   1:  PR[91,2] = PR[90,2] + 11.921;
   1:L PR[91] R[100]mm/sec CNT100;
   1:  PR[91,1] = PR[90,1] + -55.817;
   1:  PR[91,2] = PR[90,2] + 11.419;
   1:L PR[91] R[100]mm/sec CNT100;
   1:  PR[91,1] = PR[90,1] + -55.517;
   1:  PR[91,2] = PR[90,2] + 10.784;
   1:L PR[91] R[100]mm/sec CNT100;
   1:  PR[91,1] = PR[90,1] + -55.501;
   1:  PR[91,2] = PR[90,2] + 10.726;
   1:L PR[91] R[100]mm/sec CNT100;
   1:  PR[91,1] = PR[90,1] + -54.925;
   1:  PR[91,2] = PR[90,2] + 10.182;
   1:L PR[91] R[100]mm/sec CNT100;
   1:  PR[91,1] = PR[90,1] + -54.832;
   1:  PR[91,2] = PR[90,2] + 9.653;
   1:L PR[91] R[100]mm/sec CNT100;
   1:  PR[91,1] = PR[90,1] + -54.444;
   1:  PR[91,2] = PR[90,2] + 8.648;
   1:L PR[91] R[100]mm/sec CNT100;
   1:  PR[91,1] = PR[90,1] + -54.411;
   1:  PR[91,2] = PR[90,2] + 8.471;
   1:L PR[91] R[100]mm/sec CNT100;
   1:  PR[91,1] = PR[90,1] + -53.977;
   1:  PR[91,2] = PR[90,2] + 7.812;
   1:L PR[91] R[100]mm/sec CNT100;
   1:  PR[91,1] = PR[90,1] + -53.950;
   1:  PR[91,2] = PR[90,2] + 7.562;
   1:L PR[91] R[100]mm/sec CNT100;
   1:  PR[91,1] = PR[90,1] + -53.710;
   1:  PR[91,2] = PR[90,2] + 6.887;
   1:L PR[91] R[100]mm/sec CNT100;
   1:  PR[91,1] = PR[90,1] + -53.581;
   1:  PR[91,2] = PR[90,2] + 5.901;
   1:L PR[91] R[100]mm/sec CNT100;
   1:  PR[91,1] = PR[90,1] + -53.473;
   1:  PR[91,2] = PR[90,2] + 5.417;
   1:L PR[91] R[100]mm/sec CNT100;
   1:  PR[91,1] = PR[90,1] + -53.442;
   1:  PR[91,2] = PR[90,2] + 4.966;
   1:L PR[91] R[100]mm/sec CNT100;
   1:  PR[91,1] = PR[90,1] + -53.316;
   1:  PR[91,2] = PR[90,2] + 4.379;
   1:L PR[91] R[100]mm/sec CNT100;
   1:  PR[91,1] = PR[90,1] + -53.302;
   1:  PR[91,2] = PR[90,2] + 4.009;
   1:L PR[91] R[100]mm/sec CNT100;
   1:  PR[91,1] = PR[90,1] + -53.207;
   1:  PR[91,2] = PR[90,2] + 3.307;
   1:L PR[91] R[100]mm/sec CNT100;
   1:  PR[91,1] = PR[90,1] + -53.165;
   1:  PR[91,2] = PR[90,2] + 2.173;
   1:L PR[91] R[100]mm/sec CNT100;
   1:  PR[91,1] = PR[90,1] + -53.173;
   1:  PR[91,2] = PR[90,2] + 1.917;
   1:L PR[91] R[100]mm/sec CNT100;
   1:  PR[91,1] = PR[90,1] + -53.240;
   1:  PR[91,2] = PR[90,2] + 0.760;
   1:L PR[91] R[100]mm/sec CNT100;
   1:  PR[91,1] = PR[90,1] + -53.353;
   1:  PR[91,2] = PR[90,2] + -0.035;
   1:L PR[91] R[100]mm/sec CNT100;
   1:  PR[91,1] = PR[90,1] + -53.396;
   1:  PR[91,2] = PR[90,2] + -0.473;
   1:L PR[91] R[100]mm/sec CNT100;
   1:  PR[91,1] = PR[90,1] + -53.528;
   1:  PR[91,2] = PR[90,2] + -1.127;
   1:L PR[91] R[100]mm/sec CNT100;
   1:  PR[91,1] = PR[90,1] + -53.622;
   1:  PR[91,2] = PR[90,2] + -1.751;
   1:L PR[91] R[100]mm/sec CNT100;
   1:  PR[91,1] = PR[90,1] + -53.730;
   1:  PR[91,2] = PR[90,2] + -2.252;
   1:L PR[91] R[100]mm/sec CNT100;
   1:  PR[91,1] = PR[90,1] + -54.082;
   1:  PR[91,2] = PR[90,2] + -3.438;
   1:L PR[91] R[100]mm/sec CNT100;
   1:  PR[91,1] = PR[90,1] + -54.607;
   1:  PR[91,2] = PR[90,2] + -4.510;
   1:L PR[91] R[100]mm/sec CNT100;
   1:  PR[91,1] = PR[90,1] + -55.042;
   1:  PR[91,2] = PR[90,2] + -5.607;
   1:L PR[91] R[100]mm/sec CNT100;
   1:  PR[92] = PR[91];
   1:  PR[92,3] = PR[92,3] + R[101];
   1:J PR[92] R[102]% CNT100;
   1:  PR[91,1] = PR[90,1] + -50.789;
   1:  PR[91,2] = PR[90,2] + -0.113;
   1:  PR[92] = PR[91];
   1:  PR[92,3] = PR[92,3] + R[101];
   1:J PR[92] R[102]% CNT100;
   1:L PR[91] 100mm/sec CNT100 RampTo R[100];
   1:  PR[91,1] = PR[90,1] + -43.436;
   1:  PR[91,2] = PR[90,2] + 7.239;
   1:L PR[91] R[100]mm/sec CNT100;
   1:  PR[91,1] = PR[90,1] + -43.681;
   1:  PR[91,2] = PR[90,2] + 7.608;
   1:L PR[91] R[100]mm/sec CNT100;
   1:  PR[91,1] = PR[90,1] + -44.697;
   1:  PR[91,2] = PR[90,2] + 8.101;
   1:L PR[91] R[100]mm/sec CNT100;
   1:  PR[91,1] = PR[90,1] + -45.153;
   1:  PR[91,2] = PR[90,2] + 9.127;
   1:L PR[91] R[100]mm/sec CNT100;
   1:  PR[91,1] = PR[90,1] + -45.528;
   1:  PR[91,2] = PR[90,2] + 9.390;
   1:L PR[91] R[100]mm/sec CNT100;
   1:  PR[91,1] = PR[90,1] + -50.750;
   1:  PR[91,2] = PR[90,2] + 4.168;
   1:L PR[91] R[100]mm/sec CNT100;
   1:  PR[91,1] = PR[90,1] + -50.758;
   1:  PR[91,2] = PR[90,2] + 4.229;
   1:L PR[91] R[100]mm/sec CNT100;
   1:  PR[91,1] = PR[90,1] + -50.777;
   1:  PR[91,2] = PR[90,2] + 4.699;
   1:L PR[91] R[100]mm/sec CNT100;
   1:  PR[91,1] = PR[90,1] + -50.910;
   1:  PR[91,2] = PR[90,2] + 5.321;
   1:L PR[91] R[100]mm/sec CNT100;
   1:  PR[91,1] = PR[90,1] + -50.942;
   1:  PR[91,2] = PR[90,2] + 5.783;
   1:L PR[91] R[100]mm/sec CNT100;
   1:  PR[91,1] = PR[90,1] + -51.067;
   1:  PR[91,2] = PR[90,2] + 6.345;
   1:L PR[91] R[100]mm/sec CNT100;
   1:  PR[91,1] = PR[90,1] + -51.216;
   1:  PR[91,2] = PR[90,2] + 7.487;
   1:L PR[91] R[100]mm/sec CNT100;
   1:  PR[91,1] = PR[90,1] + -51.337;
   1:  PR[91,2] = PR[90,2] + 7.824;
   1:L PR[91] R[100]mm/sec CNT100;
   1:  PR[91,1] = PR[90,1] + -47.237;
   1:  PR[91,2] = PR[90,2] + 11.924;
   1:L PR[91] R[100]mm/sec CNT100;
   1:  PR[91,1] = PR[90,1] + -47.264;
   1:  PR[91,2] = PR[90,2] + 11.958;
   1:L PR[91] R[100]mm/sec CNT100;
   1:  PR[91,1] = PR[90,1] + -47.506;
   1:  PR[91,2] = PR[90,2] + 12.558;
   1:L PR[91] R[100]mm/sec CNT100;
   1:  PR[91,1] = PR[90,1] + -47.796;
   1:  PR[91,2] = PR[90,2] + 12.828;
   1:L PR[91] R[100]mm/sec CNT100;
   1:  PR[91,1] = PR[90,1] + -48.396;
   1:  PR[91,2] = PR[90,2] + 14.064;
   1:L PR[91] R[100]mm/sec CNT100;
   1:  PR[91,1] = PR[90,1] + -48.437;
   1:  PR[91,2] = PR[90,2] + 14.137;
   1:L PR[91] R[100]mm/sec CNT100;
   1:  PR[91,1] = PR[90,1] + -48.855;
   1:  PR[91,2] = PR[90,2] + 14.549;
   1:L PR[91] R[100]mm/sec CNT100;
   1:  PR[91,1] = PR[90,1] + -52.468;
   1:  PR[91,2] = PR[90,2] + 10.936;
   1:L PR[91] R[100]mm/sec CNT100;
   1:  PR[91,1] = PR[90,1] + -52.558;
   1:  PR[91,2] = PR[90,2] + 11.455;
   1:L PR[91] R[100]mm/sec CNT100;
   1:  PR[91,1] = PR[90,1] + -53.380;
   1:  PR[91,2] = PR[90,2] + 12.230;
   1:L PR[91] R[100]mm/sec CNT100;
   1:  PR[91,1] = PR[90,1] + -53.611;
   1:  PR[91,2] = PR[90,2] + 12.720;
   1:L PR[91] R[100]mm/sec CNT100;
   1:  PR[91,1] = PR[90,1] + -53.815;
   1:  PR[91,2] = PR[90,2] + 13.003;
   1:L PR[91] R[100]mm/sec CNT100;
   1:  PR[91,1] = PR[90,1] + -53.874;
   1:  PR[91,2] = PR[90,2] + 13.251;
   1:L PR[91] R[100]mm/sec CNT100;
   1:  PR[91,1] = PR[90,1] + -54.126;
   1:  PR[91,2] = PR[90,2] + 13.521;
   1:L PR[91] R[100]mm/sec CNT100;
   1:  PR[91,1] = PR[90,1] + -50.744;
   1:  PR[91,2] = PR[90,2] + 16.902;
   1:L PR[91] R[100]mm/sec CNT100;
   1:  PR[91,1] = PR[90,1] + -50.969;
   1:  PR[91,2] = PR[90,2] + 17.094;
   1:L PR[91] R[100]mm/sec CNT100;
   1:  PR[91,1] = PR[90,1] + -51.043;
   1:  PR[91,2] = PR[90,2] + 17.364;
   1:L PR[91] R[100]mm/sec CNT100;
   1:  PR[91,1] = PR[90,1] + -51.287;
   1:  PR[91,2] = PR[90,2] + 17.641;
   1:L PR[91] R[100]mm/sec CNT100;
   1:  PR[91,1] = PR[90,1] + -51.665;
   1:  PR[91,2] = PR[90,2] + 17.995;
   1:L PR[91] R[100]mm/sec CNT100;
   1:  PR[91,1] = PR[90,1] + -51.670;
   1:  PR[91,2] = PR[90,2] + 17.996;
   1:L PR[91] R[100]mm/sec CNT100;
   1:  PR[91,1] = PR[90,1] + -51.696;
   1:  PR[91,2] = PR[90,2] + 18.024;
   1:L PR[91] R[100]mm/sec CNT100;
   1:  PR[91,1] = PR[90,1] + -51.866;
   1:  PR[91,2] = PR[90,2] + 18.183;
   1:L PR[91] R[100]mm/sec CNT100;
   1:  PR[91,1] = PR[90,1] + -51.876;
   1:  PR[91,2] = PR[90,2] + 18.217;
   1:L PR[91] R[100]mm/sec CNT100;
   1:  PR[91,1] = PR[90,1] + -52.216;
   1:  PR[91,2] = PR[90,2] + 18.582;
   1:L PR[91] R[100]mm/sec CNT100;
   1:  PR[91,1] = PR[90,1] + -52.518;
   1:  PR[91,2] = PR[90,2] + 18.855;
   1:L PR[91] R[100]mm/sec CNT100;
   1:  PR[91,1] = PR[90,1] + -52.726;
   1:  PR[91,2] = PR[90,2] + 18.913;
   1:L PR[91] R[100]mm/sec CNT100;
   1:  PR[91,1] = PR[90,1] + -52.842;
   1:  PR[91,2] = PR[90,2] + 19.047;
   1:L PR[91] R[100]mm/sec CNT100;
   1:  PR[91,1] = PR[90,1] + -55.983;
   1:  PR[91,2] = PR[90,2] + 15.906;
   1:L PR[91] R[100]mm/sec CNT100;
   1:  PR[91,1] = PR[90,1] + -56.289;
   1:  PR[91,2] = PR[90,2] + 16.681;
   1:L PR[91] R[100]mm/sec CNT100;
   1:  PR[91,1] = PR[90,1] + -57.214;
   1:  PR[91,2] = PR[90,2] + 16.993;
   1:L PR[91] R[100]mm/sec CNT100;
   1:  PR[91,1] = PR[90,1] + -57.569;
   1:  PR[91,2] = PR[90,2] + 17.819;
   1:L PR[91] R[100]mm/sec CNT100;
   1:  PR[91,1] = PR[90,1] + -58.171;
   1:  PR[91,2] = PR[90,2] + 17.960;
   1:L PR[91] R[100]mm/sec CNT100;
   1:  PR[91,1] = PR[90,1] + -55.218;
   1:  PR[91,2] = PR[90,2] + 20.914;
   1:L PR[91] R[100]mm/sec CNT100;
   1:  PR[91,1] = PR[90,1] + -55.714;
   1:  PR[91,2] = PR[90,2] + 21.543;
   1:L PR[91] R[100]mm/sec CNT100;
   1:  PR[91,1] = PR[90,1] + -56.038;
   1:  PR[91,2] = PR[90,2] + 21.710;
   1:L PR[91] R[100]mm/sec CNT100;
   1:  PR[91,1] = PR[90,1] + -56.949;
   1:  PR[91,2] = PR[90,2] + 22.456;
   1:L PR[91] R[100]mm/sec CNT100;
   1:  PR[91,1] = PR[90,1] + -57.691;
   1:  PR[91,2] = PR[90,2] + 22.684;
   1:L PR[91] R[100]mm/sec CNT100;
   1:  PR[91,1] = PR[90,1] + -60.944;
   1:  PR[91,2] = PR[90,2] + 19.430;
   1:L PR[91] R[100]mm/sec CNT100;
   1:  PR[91,1] = PR[90,1] + -61.398;
   1:  PR[91,2] = PR[90,2] + 19.542;
   1:L PR[91] R[100]mm/sec CNT100;
   1:  PR[91,1] = PR[90,1] + -62.090;
   1:  PR[91,2] = PR[90,2] + 19.949;
   1:L PR[91] R[100]mm/sec CNT100;
   1:  PR[91,1] = PR[90,1] + -62.103;
   1:  PR[91,2] = PR[90,2] + 19.952;
   1:L PR[91] R[100]mm/sec CNT100;
   1:  PR[91,1] = PR[90,1] + -62.896;
   1:  PR[91,2] = PR[90,2] + 20.448;
   1:L PR[91] R[100]mm/sec CNT100;
   1:  PR[91,1] = PR[90,1] + -63.760;
   1:  PR[91,2] = PR[90,2] + 20.570;
   1:L PR[91] R[100]mm/sec CNT100;
   1:  PR[91,1] = PR[90,1] + -63.989;
   1:  PR[91,2] = PR[90,2] + 20.627;
   1:L PR[91] R[100]mm/sec CNT100;
   1:  PR[91,1] = PR[90,1] + -60.295;
   1:  PR[91,2] = PR[90,2] + 24.322;
   1:L PR[91] R[100]mm/sec CNT100;
   1:  PR[91,1] = PR[90,1] + -60.361;
   1:  PR[91,2] = PR[90,2] + 24.345;
   1:L PR[91] R[100]mm/sec CNT100;
   1:  PR[91,1] = PR[90,1] + -60.751;
   1:  PR[91,2] = PR[90,2] + 24.518;
   1:L PR[91] R[100]mm/sec CNT100;
   1:  PR[91,1] = PR[90,1] + -61.339;
   1:  PR[91,2] = PR[90,2] + 24.637;
   1:L PR[91] R[100]mm/sec CNT100;
   1:  PR[91,1] = PR[90,1] + -61.953;
   1:  PR[91,2] = PR[90,2] + 25.130;
   1:L PR[91] R[100]mm/sec CNT100;
   1:  PR[91,1] = PR[90,1] + -62.138;
   1:  PR[91,2] = PR[90,2] + 25.198;
   1:L PR[91] R[100]mm/sec CNT100;
   1:  PR[91,1] = PR[90,1] + -62.374;
   1:  PR[91,2] = PR[90,2] + 25.259;
   1:L PR[91] R[100]mm/sec CNT100;
   1:  PR[91,1] = PR[90,1] + -62.977;
   1:  PR[91,2] = PR[90,2] + 25.363;
   1:L PR[91] R[100]mm/sec CNT100;
   1:  PR[91,1] = PR[90,1] + -63.330;
   1:  PR[91,2] = PR[90,2] + 25.530;
   1:L PR[91] R[100]mm/sec CNT100;
   1:  PR[91,1] = PR[90,1] + -67.437;
   1:  PR[91,2] = PR[90,2] + 21.422;
   1:L PR[91] R[100]mm/sec CNT100;
   1:  PR[91,1] = PR[90,1] + -68.015;
   1:  PR[91,2] = PR[90,2] + 21.510;
   1:L PR[91] R[100]mm/sec CNT100;
   1:  PR[91,1] = PR[90,1] + -69.314;
   1:  PR[91,2] = PR[90,2] + 21.578;
   1:L PR[91] R[100]mm/sec CNT100;
   1:  PR[91,1] = PR[90,1] + -70.819;
   1:  PR[91,2] = PR[90,2] + 21.550;
   1:L PR[91] R[100]mm/sec CNT100;
   1:  PR[91,1] = PR[90,1] + -71.638;
   1:  PR[91,2] = PR[90,2] + 21.464;
   1:L PR[91] R[100]mm/sec CNT100;
   1:  PR[91,1] = PR[90,1] + -66.662;
   1:  PR[91,2] = PR[90,2] + 26.440;
   1:L PR[91] R[100]mm/sec CNT100;
   1:  PR[91,1] = PR[90,1] + -67.388;
   1:  PR[91,2] = PR[90,2] + 26.622;
   1:L PR[91] R[100]mm/sec CNT100;
   1:  PR[91,1] = PR[90,1] + -67.504;
   1:  PR[91,2] = PR[90,2] + 26.666;
   1:L PR[91] R[100]mm/sec CNT100;
   1:  PR[91,1] = PR[90,1] + -67.813;
   1:  PR[91,2] = PR[90,2] + 26.733;
   1:L PR[91] R[100]mm/sec CNT100;
   1:  PR[91,1] = PR[90,1] + -67.891;
   1:  PR[91,2] = PR[90,2] + 26.736;
   1:L PR[91] R[100]mm/sec CNT100;
   1:  PR[91,1] = PR[90,1] + -68.520;
   1:  PR[91,2] = PR[90,2] + 26.812;
   1:L PR[91] R[100]mm/sec CNT100;
   1:  PR[91,1] = PR[90,1] + -69.240;
   1:  PR[91,2] = PR[90,2] + 26.839;
   1:L PR[91] R[100]mm/sec CNT100;
   1:  PR[91,1] = PR[90,1] + -70.426;
   1:  PR[91,2] = PR[90,2] + 26.834;
   1:L PR[91] R[100]mm/sec CNT100;
   1:  PR[91,1] = PR[90,1] + -70.517;
   1:  PR[91,2] = PR[90,2] + 26.828;
   1:L PR[91] R[100]mm/sec CNT100;
   1:  PR[91,1] = PR[90,1] + -77.438;
   1:  PR[91,2] = PR[90,2] + 19.907;
   1:L PR[91] R[100]mm/sec CNT100;
   1:  PR[92] = PR[91];
   1:  PR[92,3] = PR[92,3] + R[101];
   1:J PR[92] R[102]% CNT100;
   1:  PR[91,1] = PR[90,1] + -91.029;
   1:  PR[91,2] = PR[90,2] + 44.499;
   1:  PR[92] = PR[91];
   1:  PR[92,3] = PR[92,3] + R[101];
   1:J PR[92] R[102]% CNT100;
   1:L PR[91] 100mm/sec CNT100 RampTo R[100];
   1:  PR[91,1] = PR[90,1] + -94.000;
   1:  PR[91,2] = PR[90,2] + 41.528;
   1:L PR[91] R[100]mm/sec CNT100;
   1:  PR[91,1] = PR[90,1] + -94.012;
   1:  PR[91,2] = PR[90,2] + 41.407;
   1:L PR[91] R[100]mm/sec CNT100;
   1:  PR[91,1] = PR[90,1] + -94.020;
   1:  PR[91,2] = PR[90,2] + 40.590;
   1:L PR[91] R[100]mm/sec CNT100;
   1:  PR[91,2] = PR[90,2] + 37.266;
   1:L PR[91] R[100]mm/sec CNT100;
   1:  PR[91,1] = PR[90,1] + -88.734;
   1:  PR[91,2] = PR[90,2] + 42.552;
   1:L PR[91] R[100]mm/sec CNT100;
   1:  PR[91,1] = PR[90,1] + -88.492;
   1:  PR[91,2] = PR[90,2] + 41.711;
   1:L PR[91] R[100]mm/sec CNT100;
   1:  PR[91,1] = PR[90,1] + -88.476;
   1:  PR[91,2] = PR[90,2] + 41.569;
   1:L PR[91] R[100]mm/sec CNT100;
   1:  PR[91,1] = PR[90,1] + -88.460;
   1:  PR[91,2] = PR[90,2] + 40.579;
   1:L PR[91] R[100]mm/sec CNT100;
   1:  PR[91,2] = PR[90,2] + 38.583;
   1:L PR[91] R[100]mm/sec CNT100;
   1:  PR[91,1] = PR[90,1] + -94.020;
   1:  PR[91,2] = PR[90,2] + 33.023;
   1:L PR[91] R[100]mm/sec CNT100;
   1:  PR[91,2] = PR[90,2] + 28.780;
   1:L PR[91] R[100]mm/sec CNT100;
   1:  PR[91,1] = PR[90,1] + -88.459;
   1:  PR[91,2] = PR[90,2] + 34.341;
   1:L PR[91] R[100]mm/sec CNT100;
   1:  PR[91,2] = PR[90,2] + 30.473;
   1:L PR[91] R[100]mm/sec CNT100;
   1:  PR[91,1] = PR[90,1] + -88.455;
   1:  PR[91,2] = PR[90,2] + 30.103;
   1:L PR[91] R[100]mm/sec CNT100;
   1:  PR[91,1] = PR[90,1] + -94.020;
   1:  PR[91,2] = PR[90,2] + 24.538;
   1:L PR[91] R[100]mm/sec CNT100;
   1:  PR[91,2] = PR[90,2] + 20.295;
   1:L PR[91] R[100]mm/sec CNT100;
   1:  PR[91,1] = PR[90,1] + -88.039;
   1:  PR[91,2] = PR[90,2] + 26.276;
   1:L PR[91] R[100]mm/sec CNT100;
   1:  PR[91,1] = PR[90,1] + -87.860;
   1:  PR[91,2] = PR[90,2] + 25.830;
   1:L PR[91] R[100]mm/sec CNT100;
   1:  PR[91,1] = PR[90,1] + -86.695;
   1:  PR[91,2] = PR[90,2] + 23.389;
   1:L PR[91] R[100]mm/sec CNT100;
   1:  PR[91,1] = PR[90,1] + -86.685;
   1:  PR[91,2] = PR[90,2] + 23.387;
   1:L PR[91] R[100]mm/sec CNT100;
   1:  PR[91,1] = PR[90,1] + -94.020;
   1:  PR[91,2] = PR[90,2] + 16.053;
   1:L PR[91] R[100]mm/sec CNT100;
   1:  PR[91,2] = PR[90,2] + 11.810;
   1:L PR[91] R[100]mm/sec CNT100;
   1:  PR[91,1] = PR[90,1] + -82.746;
   1:  PR[91,2] = PR[90,2] + 23.084;
   1:L PR[91] R[100]mm/sec CNT100;
   1:  PR[91,1] = PR[90,1] + -81.038;
   1:  PR[91,2] = PR[90,2] + 23.676;
   1:L PR[91] R[100]mm/sec CNT100;
   1:  PR[91,1] = PR[90,1] + -79.810;
   1:  PR[91,2] = PR[90,2] + 24.363;
   1:L PR[91] R[100]mm/sec CNT100;
   1:  PR[91,1] = PR[90,1] + -78.890;
   1:  PR[91,2] = PR[90,2] + 24.772;
   1:L PR[91] R[100]mm/sec CNT100;
   1:  PR[91,1] = PR[90,1] + -78.115;
   1:  PR[91,2] = PR[90,2] + 25.160;
   1:L PR[91] R[100]mm/sec CNT100;
   1:  PR[91,1] = PR[90,1] + -77.291;
   1:  PR[91,2] = PR[90,2] + 25.407;
   1:L PR[91] R[100]mm/sec CNT100;
   1:  PR[91,1] = PR[90,1] + -76.346;
   1:  PR[91,2] = PR[90,2] + 25.776;
   1:L PR[91] R[100]mm/sec CNT100;
   1:  PR[91,1] = PR[90,1] + -76.324;
   1:  PR[91,2] = PR[90,2] + 25.787;
   1:L PR[91] R[100]mm/sec CNT100;
   1:  PR[91,1] = PR[90,1] + -75.661;
   1:  PR[91,2] = PR[90,2] + 26.005;
   1:L PR[91] R[100]mm/sec CNT100;
   1:  PR[91,1] = PR[90,1] + -75.568;
   1:  PR[91,2] = PR[90,2] + 26.019;
   1:L PR[91] R[100]mm/sec CNT100;
   1:  PR[91,1] = PR[90,1] + -94.020;
   1:  PR[91,2] = PR[90,2] + 7.568;
   1:L PR[91] R[100]mm/sec CNT100;
   1:  PR[91,1] = PR[90,1] + -94.019;
   1:  PR[91,2] = PR[90,2] + 3.325;
   1:L PR[91] R[100]mm/sec CNT100;
   1:  PR[91,1] = PR[90,1] + -87.134;
   1:  PR[91,2] = PR[90,2] + 10.211;
   1:L PR[91] R[100]mm/sec CNT100;
   1:  PR[91,1] = PR[90,1] + -87.246;
   1:  PR[91,2] = PR[90,2] + 9.982;
   1:L PR[91] R[100]mm/sec CNT100;
   1:  PR[91,1] = PR[90,1] + -87.849;
   1:  PR[91,2] = PR[90,2] + 8.500;
   1:L PR[91] R[100]mm/sec CNT100;
   1:  PR[91,1] = PR[90,1] + -88.076;
   1:  PR[91,2] = PR[90,2] + 7.623;
   1:L PR[91] R[100]mm/sec CNT100;
   1:  PR[91,1] = PR[90,1] + -88.169;
   1:  PR[91,2] = PR[90,2] + 7.136;
   1:L PR[91] R[100]mm/sec CNT100;
   1:  PR[91,1] = PR[90,1] + -88.449;
   1:  PR[91,2] = PR[90,2] + 6.125;
   1:L PR[91] R[100]mm/sec CNT100;
   1:  PR[91,1] = PR[90,1] + -88.473;
   1:  PR[91,2] = PR[90,2] + 5.861;
   1:L PR[91] R[100]mm/sec CNT100;
   1:  PR[91,1] = PR[90,1] + -88.707;
   1:  PR[91,2] = PR[90,2] + 4.884;
   1:L PR[91] R[100]mm/sec CNT100;
   1:  PR[91,1] = PR[90,1] + -88.766;
   1:  PR[91,2] = PR[90,2] + 4.336;
   1:L PR[91] R[100]mm/sec CNT100;
   1:  PR[91,1] = PR[90,1] + -93.775;
   1:  PR[91,2] = PR[90,2] + -0.673;
   1:L PR[91] R[100]mm/sec CNT100;
   1:  PR[91,1] = PR[90,1] + -93.743;
   1:  PR[91,2] = PR[90,2] + -0.817;
   1:L PR[91] R[100]mm/sec CNT100;
   1:  PR[91,1] = PR[90,1] + -93.466;
   1:  PR[91,2] = PR[90,2] + -2.169;
   1:L PR[91] R[100]mm/sec CNT100;
   1:  PR[91,1] = PR[90,1] + -93.454;
   1:  PR[91,2] = PR[90,2] + -2.408;
   1:L PR[91] R[100]mm/sec CNT100;
   1:  PR[91,1] = PR[90,1] + -93.353;
   1:  PR[91,2] = PR[90,2] + -2.936;
   1:L PR[91] R[100]mm/sec CNT100;
   1:  PR[91,1] = PR[90,1] + -93.260;
   1:  PR[91,2] = PR[90,2] + -3.724;
   1:L PR[91] R[100]mm/sec CNT100;
   1:  PR[91,1] = PR[90,1] + -93.149;
   1:  PR[91,2] = PR[90,2] + -4.167;
   1:L PR[91] R[100]mm/sec CNT100;
   1:  PR[91,1] = PR[90,1] + -93.138;
   1:  PR[91,2] = PR[90,2] + -4.257;
   1:L PR[91] R[100]mm/sec CNT100;
   1:  PR[91,1] = PR[90,1] + -93.131;
   1:  PR[91,2] = PR[90,2] + -4.272;
   1:L PR[91] R[100]mm/sec CNT100;
   1:  PR[91,1] = PR[90,1] + -88.764;
   1:  PR[91,2] = PR[90,2] + 0.096;
   1:L PR[91] R[100]mm/sec CNT100;
   1:  PR[91,1] = PR[90,1] + -88.650;
   1:  PR[91,2] = PR[90,2] + -0.773;
   1:L PR[91] R[100]mm/sec CNT100;
   1:  PR[91,1] = PR[90,1] + -88.448;
   1:  PR[91,2] = PR[90,2] + -1.417;
   1:L PR[91] R[100]mm/sec CNT100;
   1:  PR[91,1] = PR[90,1] + -88.428;
   1:  PR[91,2] = PR[90,2] + -1.723;
   1:L PR[91] R[100]mm/sec CNT100;
   1:  PR[91,1] = PR[90,1] + -88.200;
   1:  PR[91,2] = PR[90,2] + -2.336;
   1:L PR[91] R[100]mm/sec CNT100;
   1:  PR[91,1] = PR[90,1] + -88.175;
   1:  PR[91,2] = PR[90,2] + -2.645;
   1:L PR[91] R[100]mm/sec CNT100;
   1:  PR[91,1] = PR[90,1] + -87.988;
   1:  PR[91,2] = PR[90,2] + -3.260;
   1:L PR[91] R[100]mm/sec CNT100;
   1:  PR[91,1] = PR[90,1] + -87.970;
   1:  PR[91,2] = PR[90,2] + -3.353;
   1:L PR[91] R[100]mm/sec CNT100;
   1:  PR[91,1] = PR[90,1] + -91.962;
   1:  PR[91,2] = PR[90,2] + -7.345;
   1:L PR[91] R[100]mm/sec CNT100;
   1:  PR[91,1] = PR[90,1] + -91.533;
   1:  PR[91,2] = PR[90,2] + -8.166;
   1:L PR[91] R[100]mm/sec CNT100;
   1:  PR[91,1] = PR[90,1] + -91.398;
   1:  PR[91,2] = PR[90,2] + -8.701;
   1:L PR[91] R[100]mm/sec CNT100;
   1:  PR[91,1] = PR[90,1] + -91.349;
   1:  PR[91,2] = PR[90,2] + -8.776;
   1:L PR[91] R[100]mm/sec CNT100;
   1:  PR[91,1] = PR[90,1] + -90.903;
   1:  PR[91,2] = PR[90,2] + -9.411;
   1:L PR[91] R[100]mm/sec CNT100;
   1:  PR[91,1] = PR[90,1] + -90.892;
   1:  PR[91,2] = PR[90,2] + -9.482;
   1:L PR[91] R[100]mm/sec CNT100;
   1:  PR[91,1] = PR[90,1] + -90.650;
   1:  PR[91,2] = PR[90,2] + -9.854;
   1:L PR[91] R[100]mm/sec CNT100;
   1:  PR[91,1] = PR[90,1] + -90.594;
   1:  PR[91,2] = PR[90,2] + -10.020;
   1:L PR[91] R[100]mm/sec CNT100;
   1:  PR[91,1] = PR[90,1] + -90.477;
   1:  PR[91,2] = PR[90,2] + -10.103;
   1:L PR[91] R[100]mm/sec CNT100;
   1:  PR[91,1] = PR[90,1] + -86.782;
   1:  PR[91,2] = PR[90,2] + -6.408;
   1:L PR[91] R[100]mm/sec CNT100;
   1:  PR[91,1] = PR[90,1] + -86.570;
   1:  PR[91,2] = PR[90,2] + -7.052;
   1:L PR[91] R[100]mm/sec CNT100;
   1:  PR[91,1] = PR[90,1] + -86.168;
   1:  PR[91,2] = PR[90,2] + -7.616;
   1:L PR[91] R[100]mm/sec CNT100;
   1:  PR[91,1] = PR[90,1] + -86.145;
   1:  PR[91,2] = PR[90,2] + -7.724;
   1:L PR[91] R[100]mm/sec CNT100;
   1:  PR[91,1] = PR[90,1] + -85.725;
   1:  PR[91,2] = PR[90,2] + -8.237;
   1:L PR[91] R[100]mm/sec CNT100;
   1:  PR[91,1] = PR[90,1] + -85.499;
   1:  PR[91,2] = PR[90,2] + -8.554;
   1:L PR[91] R[100]mm/sec CNT100;
   1:  PR[91,1] = PR[90,1] + -85.301;
   1:  PR[91,2] = PR[90,2] + -9.169;
   1:L PR[91] R[100]mm/sec CNT100;
   1:  PR[91,1] = PR[90,1] + -88.798;
   1:  PR[91,2] = PR[90,2] + -12.667;
   1:L PR[91] R[100]mm/sec CNT100;
   1:  PR[91,1] = PR[90,1] + -88.790;
   1:  PR[91,2] = PR[90,2] + -12.686;
   1:L PR[91] R[100]mm/sec CNT100;
   1:  PR[91,1] = PR[90,1] + -88.096;
   1:  PR[91,2] = PR[90,2] + -13.131;
   1:L PR[91] R[100]mm/sec CNT100;
   1:  PR[91,1] = PR[90,1] + -87.921;
   1:  PR[91,2] = PR[90,2] + -13.611;
   1:L PR[91] R[100]mm/sec CNT100;
   1:  PR[91,1] = PR[90,1] + -87.266;
   1:  PR[91,2] = PR[90,2] + -13.909;
   1:L PR[91] R[100]mm/sec CNT100;
   1:  PR[91,1] = PR[90,1] + -87.043;
   1:  PR[91,2] = PR[90,2] + -14.534;
   1:L PR[91] R[100]mm/sec CNT100;
   1:  PR[91,1] = PR[90,1] + -86.595;
   1:  PR[91,2] = PR[90,2] + -14.706;
   1:L PR[91] R[100]mm/sec CNT100;
   1:  PR[91,1] = PR[90,1] + -83.282;
   1:  PR[91,2] = PR[90,2] + -11.393;
   1:L PR[91] R[100]mm/sec CNT100;
   1:  PR[91,1] = PR[90,1] + -83.104;
   1:  PR[91,2] = PR[90,2] + -11.497;
   1:L PR[91] R[100]mm/sec CNT100;
   1:  PR[91,1] = PR[90,1] + -82.606;
   1:  PR[91,2] = PR[90,2] + -12.329;
   1:L PR[91] R[100]mm/sec CNT100;
   1:  PR[91,1] = PR[90,1] + -81.683;
   1:  PR[91,2] = PR[90,2] + -12.735;
   1:L PR[91] R[100]mm/sec CNT100;
   1:  PR[91,1] = PR[90,1] + -81.336;
   1:  PR[91,2] = PR[90,2] + -13.191;
   1:L PR[91] R[100]mm/sec CNT100;
   1:  PR[91,1] = PR[90,1] + -81.009;
   1:  PR[91,2] = PR[90,2] + -13.362;
   1:L PR[91] R[100]mm/sec CNT100;
   1:  PR[91,1] = PR[90,1] + -84.506;
   1:  PR[91,2] = PR[90,2] + -16.860;
   1:L PR[91] R[100]mm/sec CNT100;
   1:  PR[91,1] = PR[90,1] + -84.265;
   1:  PR[91,2] = PR[90,2] + -17.222;
   1:L PR[91] R[100]mm/sec CNT100;
   1:  PR[91,1] = PR[90,1] + -84.025;
   1:  PR[91,2] = PR[90,2] + -17.343;
   1:L PR[91] R[100]mm/sec CNT100;
   1:  PR[91,1] = PR[90,1] + -83.231;
   1:  PR[91,2] = PR[90,2] + -18.021;
   1:L PR[91] R[100]mm/sec CNT100;
   1:  PR[91,1] = PR[90,1] + -83.176;
   1:  PR[91,2] = PR[90,2] + -18.064;
   1:L PR[91] R[100]mm/sec CNT100;
   1:  PR[91,1] = PR[90,1] + -82.265;
   1:  PR[91,2] = PR[90,2] + -18.281;
   1:L PR[91] R[100]mm/sec CNT100;
   1:  PR[91,1] = PR[90,1] + -81.993;
   1:  PR[91,2] = PR[90,2] + -18.589;
   1:L PR[91] R[100]mm/sec CNT100;
   1:  PR[91,1] = PR[90,1] + -78.384;
   1:  PR[91,2] = PR[90,2] + -14.980;
   1:L PR[91] R[100]mm/sec CNT100;
   1:  PR[91,1] = PR[90,1] + -77.519;
   1:  PR[91,2] = PR[90,2] + -15.217;
   1:L PR[91] R[100]mm/sec CNT100;
   1:  PR[91,1] = PR[90,1] + -76.865;
   1:  PR[91,2] = PR[90,2] + -15.557;
   1:L PR[91] R[100]mm/sec CNT100;
   1:  PR[91,1] = PR[90,1] + -76.139;
   1:  PR[91,2] = PR[90,2] + -15.998;
   1:L PR[91] R[100]mm/sec CNT100;
   1:  PR[91,1] = PR[90,1] + -75.487;
   1:  PR[91,2] = PR[90,2] + -16.102;
   1:L PR[91] R[100]mm/sec CNT100;
   1:  PR[91,1] = PR[90,1] + -75.314;
   1:  PR[91,2] = PR[90,2] + -16.153;
   1:L PR[91] R[100]mm/sec CNT100;
   1:  PR[91,1] = PR[90,1] + -79.234;
   1:  PR[91,2] = PR[90,2] + -20.074;
   1:L PR[91] R[100]mm/sec CNT100;
   1:  PR[91,1] = PR[90,1] + -78.872;
   1:  PR[91,2] = PR[90,2] + -20.127;
   1:L PR[91] R[100]mm/sec CNT100;
   1:  PR[91,1] = PR[90,1] + -78.083;
   1:  PR[91,2] = PR[90,2] + -20.713;
   1:L PR[91] R[100]mm/sec CNT100;
   1:  PR[91,1] = PR[90,1] + -77.986;
   1:  PR[91,2] = PR[90,2] + -20.754;
   1:L PR[91] R[100]mm/sec CNT100;
   1:  PR[91,1] = PR[90,1] + -77.278;
   1:  PR[91,2] = PR[90,2] + -20.880;
   1:L PR[91] R[100]mm/sec CNT100;
   1:  PR[91,1] = PR[90,1] + -76.754;
   1:  PR[91,2] = PR[90,2] + -21.055;
   1:L PR[91] R[100]mm/sec CNT100;
   1:  PR[91,1] = PR[90,1] + -76.384;
   1:  PR[91,2] = PR[90,2] + -21.092;
   1:L PR[91] R[100]mm/sec CNT100;
   1:  PR[91,1] = PR[90,1] + -76.133;
   1:  PR[91,2] = PR[90,2] + -21.214;
   1:L PR[91] R[100]mm/sec CNT100;
   1:  PR[91,1] = PR[90,1] + -71.694;
   1:  PR[91,2] = PR[90,2] + -16.776;
   1:L PR[91] R[100]mm/sec CNT100;
   1:  PR[91,1] = PR[90,1] + -71.651;
   1:  PR[91,2] = PR[90,2] + -16.778;
   1:L PR[91] R[100]mm/sec CNT100;
   1:  PR[91,1] = PR[90,1] + -70.899;
   1:  PR[91,2] = PR[90,2] + -16.880;
   1:L PR[91] R[100]mm/sec CNT100;
   1:  PR[91,1] = PR[90,1] + -69.517;
   1:  PR[91,2] = PR[90,2] + -16.917;
   1:L PR[91] R[100]mm/sec CNT100;
   1:  PR[91,1] = PR[90,1] + -67.947;
   1:  PR[91,2] = PR[90,2] + -16.839;
   1:L PR[91] R[100]mm/sec CNT100;
   1:  PR[91,1] = PR[90,1] + -67.436;
   1:  PR[91,2] = PR[90,2] + -16.760;
   1:L PR[91] R[100]mm/sec CNT100;
   1:  PR[91,1] = PR[90,1] + -72.601;
   1:  PR[91,2] = PR[90,2] + -21.925;
   1:L PR[91] R[100]mm/sec CNT100;
   1:  PR[91,1] = PR[90,1] + -72.086;
   1:  PR[91,2] = PR[90,2] + -21.999;
   1:L PR[91] R[100]mm/sec CNT100;
   1:  PR[91,1] = PR[90,1] + -71.220;
   1:  PR[91,2] = PR[90,2] + -22.087;
   1:L PR[91] R[100]mm/sec CNT100;
   1:  PR[91,1] = PR[90,1] + -70.415;
   1:  PR[91,2] = PR[90,2] + -22.147;
   1:L PR[91] R[100]mm/sec CNT100;
   1:  PR[91,1] = PR[90,1] + -69.635;
   1:  PR[91,2] = PR[90,2] + -22.162;
   1:L PR[91] R[100]mm/sec CNT100;
   1:  PR[91,1] = PR[90,1] + -68.851;
   1:  PR[91,2] = PR[90,2] + -22.119;
   1:L PR[91] R[100]mm/sec CNT100;
   1:  PR[91,1] = PR[90,1] + -68.523;
   1:  PR[91,2] = PR[90,2] + -22.090;
   1:L PR[91] R[100]mm/sec CNT100;
   1:  PR[91,1] = PR[90,1] + -61.511;
   1:  PR[91,2] = PR[90,2] + -15.078;
   1:L PR[91] R[100]mm/sec CNT100;
   1:  PR[91,1] = PR[90,1] + -60.617;
   1:  PR[91,2] = PR[90,2] + -14.709;
   1:L PR[91] R[100]mm/sec CNT100;
   1:  PR[91,1] = PR[90,1] + -58.370;
   1:  PR[91,2] = PR[90,2] + -13.214;
   1:L PR[91] R[100]mm/sec CNT100;
   1:  PR[91,1] = PR[90,1] + -57.966;
   1:  PR[91,2] = PR[90,2] + -12.872;
   1:L PR[91] R[100]mm/sec CNT100;
   1:  PR[91,1] = PR[90,1] + -56.844;
   1:  PR[91,2] = PR[90,2] + -12.000;
   1:L PR[91] R[100]mm/sec CNT100;
   1:  PR[91,1] = PR[90,1] + -55.451;
   1:  PR[91,2] = PR[90,2] + -10.598;
   1:L PR[91] R[100]mm/sec CNT100;
   1:  PR[91,1] = PR[90,1] + -54.574;
   1:  PR[91,2] = PR[90,2] + -9.450;
   1:L PR[91] R[100]mm/sec CNT100;
   1:  PR[91,1] = PR[90,1] + -54.232;
   1:  PR[91,2] = PR[90,2] + -9.033;
   1:L PR[91] R[100]mm/sec CNT100;
   1:  PR[91,1] = PR[90,1] + -52.765;
   1:  PR[91,2] = PR[90,2] + -6.785;
   1:L PR[91] R[100]mm/sec CNT100;
   1:  PR[91,1] = PR[90,1] + -52.469;
   1:  PR[91,2] = PR[90,2] + -6.036;
   1:L PR[91] R[100]mm/sec CNT100;
   1:  PR[91,1] = PR[90,1] + -40.759;
   1:  PR[91,2] = PR[90,2] + 5.674;
   1:L PR[91] R[100]mm/sec CNT100;
   1:  PR[91,1] = PR[90,1] + -40.173;
   1:  PR[91,2] = PR[90,2] + 5.261;
   1:L PR[91] R[100]mm/sec CNT100;
   1:  PR[91,1] = PR[90,1] + -39.299;
   1:  PR[91,2] = PR[90,2] + 5.102;
   1:L PR[91] R[100]mm/sec CNT100;
   1:  PR[91,1] = PR[90,1] + -38.689;
   1:  PR[91,2] = PR[90,2] + 4.938;
   1:L PR[91] R[100]mm/sec CNT100;
   1:  PR[91,1] = PR[90,1] + -37.950;
   1:  PR[91,2] = PR[90,2] + 4.791;
   1:L PR[91] R[100]mm/sec CNT100;
   1:  PR[91,1] = PR[90,1] + -37.437;
   1:  PR[91,2] = PR[90,2] + 4.753;
   1:L PR[91] R[100]mm/sec CNT100;
   1:  PR[91,1] = PR[90,1] + -63.191;
   1:  PR[91,2] = PR[90,2] + -21.000;
   1:L PR[91] R[100]mm/sec CNT100;
   1:  PR[91,1] = PR[90,1] + -62.841;
   1:  PR[91,2] = PR[90,2] + -20.903;
   1:L PR[91] R[100]mm/sec CNT100;
   1:  PR[91,1] = PR[90,1] + -62.078;
   1:  PR[91,2] = PR[90,2] + -20.590;
   1:L PR[91] R[100]mm/sec CNT100;
   1:  PR[91,1] = PR[90,1] + -61.998;
   1:  PR[91,2] = PR[90,2] + -20.571;
   1:L PR[91] R[100]mm/sec CNT100;
   1:  PR[91,1] = PR[90,1] + -61.899;
   1:  PR[91,2] = PR[90,2] + -20.516;
   1:L PR[91] R[100]mm/sec CNT100;
   1:  PR[91,1] = PR[90,1] + -61.158;
   1:  PR[91,2] = PR[90,2] + -20.182;
   1:L PR[91] R[100]mm/sec CNT100;
   1:  PR[91,1] = PR[90,1] + -60.551;
   1:  PR[91,2] = PR[90,2] + -19.916;
   1:L PR[91] R[100]mm/sec CNT100;
   1:  PR[91,1] = PR[90,1] + -60.264;
   1:  PR[91,2] = PR[90,2] + -19.816;
   1:L PR[91] R[100]mm/sec CNT100;
   1:  PR[91,1] = PR[90,1] + -59.968;
   1:  PR[91,2] = PR[90,2] + -19.632;
   1:L PR[91] R[100]mm/sec CNT100;
   1:  PR[91,1] = PR[90,1] + -59.437;
   1:  PR[91,2] = PR[90,2] + -19.337;
   1:L PR[91] R[100]mm/sec CNT100;
   1:  PR[91,1] = PR[90,1] + -58.785;
   1:  PR[91,2] = PR[90,2] + -18.992;
   1:L PR[91] R[100]mm/sec CNT100;
   1:  PR[91,1] = PR[90,1] + -58.504;
   1:  PR[91,2] = PR[90,2] + -18.869;
   1:L PR[91] R[100]mm/sec CNT100;
   1:  PR[91,1] = PR[90,1] + -58.302;
   1:  PR[91,2] = PR[90,2] + -18.725;
   1:L PR[91] R[100]mm/sec CNT100;
   1:  PR[91,1] = PR[90,1] + -57.675;
   1:  PR[91,2] = PR[90,2] + -18.346;
   1:L PR[91] R[100]mm/sec CNT100;
   1:  PR[91,1] = PR[90,1] + -56.706;
   1:  PR[91,2] = PR[90,2] + -17.692;
   1:L PR[91] R[100]mm/sec CNT100;
   1:  PR[91,1] = PR[90,1] + -55.872;
   1:  PR[91,2] = PR[90,2] + -17.164;
   1:L PR[91] R[100]mm/sec CNT100;
   1:  PR[91,1] = PR[90,1] + -55.583;
   1:  PR[91,2] = PR[90,2] + -16.924;
   1:L PR[91] R[100]mm/sec CNT100;
   1:  PR[91,1] = PR[90,1] + -55.037;
   1:  PR[91,2] = PR[90,2] + -16.506;
   1:L PR[91] R[100]mm/sec CNT100;
   1:  PR[91,1] = PR[90,1] + -54.165;
   1:  PR[91,2] = PR[90,2] + -15.752;
   1:L PR[91] R[100]mm/sec CNT100;
   1:  PR[91,1] = PR[90,1] + -53.253;
   1:  PR[91,2] = PR[90,2] + -14.918;
   1:L PR[91] R[100]mm/sec CNT100;
   1:  PR[91,1] = PR[90,1] + -52.348;
   1:  PR[91,2] = PR[90,2] + -14.032;
   1:L PR[91] R[100]mm/sec CNT100;
   1:  PR[91,1] = PR[90,1] + -51.647;
   1:  PR[91,2] = PR[90,2] + -13.295;
   1:L PR[91] R[100]mm/sec CNT100;
   1:  PR[91,1] = PR[90,1] + -50.508;
   1:  PR[91,2] = PR[90,2] + -12.023;
   1:L PR[91] R[100]mm/sec CNT100;
   1:  PR[91,1] = PR[90,1] + -50.017;
   1:  PR[91,2] = PR[90,2] + -11.444;
   1:L PR[91] R[100]mm/sec CNT100;
   1:  PR[91,1] = PR[90,1] + -49.346;
   1:  PR[91,2] = PR[90,2] + -10.604;
   1:L PR[91] R[100]mm/sec CNT100;
   1:  PR[91,1] = PR[90,1] + -48.782;
   1:  PR[91,2] = PR[90,2] + -9.771;
   1:L PR[91] R[100]mm/sec CNT100;
   1:  PR[91,1] = PR[90,1] + -48.120;
   1:  PR[91,2] = PR[90,2] + -8.734;
   1:L PR[91] R[100]mm/sec CNT100;
   1:  PR[91,1] = PR[90,1] + -47.462;
   1:  PR[91,2] = PR[90,2] + -7.792;
   1:L PR[91] R[100]mm/sec CNT100;
   1:  PR[91,1] = PR[90,1] + -46.864;
   1:  PR[91,2] = PR[90,2] + -6.764;
   1:L PR[91] R[100]mm/sec CNT100;
   1:  PR[91,1] = PR[90,1] + -45.944;
   1:  PR[91,2] = PR[90,2] + -5.472;
   1:L PR[91] R[100]mm/sec CNT100;
   1:  PR[91,1] = PR[90,1] + -44.948;
   1:  PR[91,2] = PR[90,2] + -4.281;
   1:L PR[91] R[100]mm/sec CNT100;
   1:  PR[91,1] = PR[90,1] + -44.341;
   1:  PR[91,2] = PR[90,2] + -3.608;
   1:L PR[91] R[100]mm/sec CNT100;
   1:  PR[91,1] = PR[90,1] + -43.629;
   1:  PR[91,2] = PR[90,2] + -2.917;
   1:L PR[91] R[100]mm/sec CNT100;
   1:  PR[91,1] = PR[90,1] + -42.884;
   1:  PR[91,2] = PR[90,2] + -2.293;
   1:L PR[91] R[100]mm/sec CNT100;
   1:  PR[91,1] = PR[90,1] + -41.296;
   1:  PR[91,2] = PR[90,2] + -1.183;
   1:L PR[91] R[100]mm/sec CNT100;
   1:  PR[91,1] = PR[90,1] + -39.750;
   1:  PR[91,2] = PR[90,2] + -0.622;
   1:L PR[91] R[100]mm/sec CNT100;
   1:  PR[91,1] = PR[90,1] + -38.740;
   1:  PR[91,2] = PR[90,2] + -0.280;
   1:L PR[91] R[100]mm/sec CNT100;
   1:  PR[91,1] = PR[90,1] + -38.283;
   1:  PR[91,2] = PR[90,2] + -0.192;
   1:L PR[91] R[100]mm/sec CNT100;
   1:  PR[91,1] = PR[90,1] + -38.091;
   1:  PR[91,2] = PR[90,2] + -0.144;
   1:L PR[91] R[100]mm/sec CNT100;
   1:  PR[91,1] = PR[90,1] + -33.221;
   1:  PR[91,2] = PR[90,2] + 4.727;
   1:L PR[91] R[100]mm/sec CNT100;
   1:  PR[91,1] = PR[90,1] + -32.523;
   1:  PR[91,2] = PR[90,2] + 4.845;
   1:L PR[91] R[100]mm/sec CNT100;
   1:  PR[91,1] = PR[90,1] + -31.694;
   1:  PR[91,2] = PR[90,2] + 5.065;
   1:L PR[91] R[100]mm/sec CNT100;
   1:  PR[91,1] = PR[90,1] + -31.039;
   1:  PR[91,2] = PR[90,2] + 5.197;
   1:L PR[91] R[100]mm/sec CNT100;
   1:  PR[91,1] = PR[90,1] + -30.060;
   1:  PR[91,2] = PR[90,2] + 5.694;
   1:L PR[91] R[100]mm/sec CNT100;
   1:  PR[91,1] = PR[90,1] + -29.393;
   1:  PR[91,2] = PR[90,2] + 6.086;
   1:L PR[91] R[100]mm/sec CNT100;
   1:  PR[91,1] = PR[90,1] + -28.122;
   1:  PR[91,2] = PR[90,2] + 6.764;
   1:L PR[91] R[100]mm/sec CNT100;
   1:  PR[91,1] = PR[90,1] + -26.485;
   1:  PR[91,2] = PR[90,2] + 8.087;
   1:L PR[91] R[100]mm/sec CNT100;
   1:  PR[91,1] = PR[90,1] + -26.138;
   1:  PR[91,2] = PR[90,2] + 8.353;
   1:L PR[91] R[100]mm/sec CNT100;
   1:  PR[91,1] = PR[90,1] + -25.495;
   1:  PR[91,2] = PR[90,2] + 8.708;
   1:L PR[91] R[100]mm/sec CNT100;
   1:  PR[91,1] = PR[90,1] + -24.922;
   1:  PR[91,2] = PR[90,2] + 8.984;
   1:L PR[91] R[100]mm/sec CNT100;
   1:  PR[91,1] = PR[90,1] + -24.645;
   1:  PR[91,2] = PR[90,2] + 9.060;
   1:L PR[91] R[100]mm/sec CNT100;
   1:  PR[91,1] = PR[90,1] + -33.597;
   1:  PR[91,2] = PR[90,2] + 0.108;
   1:L PR[91] R[100]mm/sec CNT100;
   1:  PR[91,1] = PR[90,1] + -32.840;
   1:  PR[91,2] = PR[90,2] + -0.122;
   1:L PR[91] R[100]mm/sec CNT100;
   1:  PR[91,1] = PR[90,1] + -32.446;
   1:  PR[91,2] = PR[90,2] + -0.155;
   1:L PR[91] R[100]mm/sec CNT100;
   1:  PR[91,1] = PR[90,1] + -31.752;
   1:  PR[91,2] = PR[90,2] + -0.432;
   1:L PR[91] R[100]mm/sec CNT100;
   1:  PR[91,1] = PR[90,1] + -31.468;
   1:  PR[91,2] = PR[90,2] + -0.477;
   1:L PR[91] R[100]mm/sec CNT100;
   1:  PR[91,1] = PR[90,1] + -30.617;
   1:  PR[91,2] = PR[90,2] + -0.736;
   1:L PR[91] R[100]mm/sec CNT100;
   1:  PR[91,1] = PR[90,1] + -30.324;
   1:  PR[91,2] = PR[90,2] + -0.862;
   1:L PR[91] R[100]mm/sec CNT100;
   1:  PR[91,1] = PR[90,1] + -20.325;
   1:  PR[91,2] = PR[90,2] + 9.138;
   1:L PR[91] R[100]mm/sec CNT100;
   1:  PR[91,1] = PR[90,1] + -20.321;
   1:  PR[91,2] = PR[90,2] + 9.136;
   1:L PR[91] R[100]mm/sec CNT100;
   1:  PR[91,1] = PR[90,1] + -20.057;
   1:  PR[91,2] = PR[90,2] + 9.108;
   1:L PR[91] R[100]mm/sec CNT100;
   1:  PR[91,1] = PR[90,1] + -19.506;
   1:  PR[91,2] = PR[90,2] + 8.960;
   1:L PR[91] R[100]mm/sec CNT100;
   1:  PR[91,1] = PR[90,1] + -19.398;
   1:  PR[91,2] = PR[90,2] + 8.894;
   1:L PR[91] R[100]mm/sec CNT100;
   1:  PR[91,1] = PR[90,1] + -18.882;
   1:  PR[91,2] = PR[90,2] + 8.524;
   1:L PR[91] R[100]mm/sec CNT100;
   1:  PR[91,1] = PR[90,1] + -18.770;
   1:  PR[91,2] = PR[90,2] + 8.506;
   1:L PR[91] R[100]mm/sec CNT100;
   1:  PR[91,1] = PR[90,1] + -18.528;
   1:  PR[91,2] = PR[90,2] + 8.357;
   1:L PR[91] R[100]mm/sec CNT100;
   1:  PR[91,1] = PR[90,1] + -18.451;
   1:  PR[91,2] = PR[90,2] + 8.323;
   1:L PR[91] R[100]mm/sec CNT100;
   1:  PR[91,1] = PR[90,1] + -18.051;
   1:  PR[91,2] = PR[90,2] + 7.811;
   1:L PR[91] R[100]mm/sec CNT100;
   1:  PR[91,1] = PR[90,1] + -17.645;
   1:  PR[91,2] = PR[90,2] + 7.627;
   1:L PR[91] R[100]mm/sec CNT100;
   1:  PR[91,1] = PR[90,1] + -17.626;
   1:  PR[91,2] = PR[90,2] + 7.594;
   1:L PR[91] R[100]mm/sec CNT100;
   1:  PR[91,1] = PR[90,1] + -27.545;
   1:  PR[91,2] = PR[90,2] + -2.325;
   1:L PR[91] R[100]mm/sec CNT100;
   1:  PR[91,1] = PR[90,1] + -26.956;
   1:  PR[91,2] = PR[90,2] + -3.024;
   1:L PR[91] R[100]mm/sec CNT100;
   1:  PR[91,1] = PR[90,1] + -26.697;
   1:  PR[91,2] = PR[90,2] + -3.184;
   1:L PR[91] R[100]mm/sec CNT100;
   1:  PR[91,1] = PR[90,1] + -26.644;
   1:  PR[91,2] = PR[90,2] + -3.224;
   1:L PR[91] R[100]mm/sec CNT100;
   1:  PR[91,1] = PR[90,1] + -26.552;
   1:  PR[91,2] = PR[90,2] + -3.244;
   1:L PR[91] R[100]mm/sec CNT100;
   1:  PR[91,1] = PR[90,1] + -25.930;
   1:  PR[91,2] = PR[90,2] + -3.751;
   1:L PR[91] R[100]mm/sec CNT100;
   1:  PR[91,1] = PR[90,1] + -25.507;
   1:  PR[91,2] = PR[90,2] + -3.852;
   1:L PR[91] R[100]mm/sec CNT100;
   1:  PR[91,1] = PR[90,1] + -25.083;
   1:  PR[91,2] = PR[90,2] + -4.106;
   1:L PR[91] R[100]mm/sec CNT100;
   1:  PR[91,1] = PR[90,1] + -15.831;
   1:  PR[91,2] = PR[90,2] + 5.146;
   1:L PR[91] R[100]mm/sec CNT100;
   1:  PR[91,1] = PR[90,1] + -15.769;
   1:  PR[91,2] = PR[90,2] + 5.016;
   1:L PR[91] R[100]mm/sec CNT100;
   1:  PR[91,1] = PR[90,1] + -15.634;
   1:  PR[91,2] = PR[90,2] + 4.849;
   1:L PR[91] R[100]mm/sec CNT100;
   1:  PR[91,1] = PR[90,1] + -15.631;
   1:  PR[91,2] = PR[90,2] + 4.837;
   1:L PR[91] R[100]mm/sec CNT100;
   1:  PR[91,1] = PR[90,1] + -15.589;
   1:  PR[91,2] = PR[90,2] + 4.613;
   1:L PR[91] R[100]mm/sec CNT100;
   1:  PR[91,1] = PR[90,1] + -15.546;
   1:  PR[91,2] = PR[90,2] + 4.221;
   1:L PR[91] R[100]mm/sec CNT100;
   1:  PR[91,1] = PR[90,1] + -15.345;
   1:  PR[91,2] = PR[90,2] + 3.396;
   1:L PR[91] R[100]mm/sec CNT100;
   1:  PR[91,1] = PR[90,1] + -15.245;
   1:  PR[91,2] = PR[90,2] + 2.758;
   1:L PR[91] R[100]mm/sec CNT100;
   1:  PR[91,1] = PR[90,1] + -15.220;
   1:  PR[91,2] = PR[90,2] + 2.661;
   1:L PR[91] R[100]mm/sec CNT100;
   1:  PR[91,1] = PR[90,1] + -15.202;
   1:  PR[91,2] = PR[90,2] + 2.260;
   1:L PR[91] R[100]mm/sec CNT100;
   1:  PR[91,1] = PR[90,1] + -15.252;
   1:  PR[91,2] = PR[90,2] + 1.721;
   1:L PR[91] R[100]mm/sec CNT100;
   1:  PR[91,1] = PR[90,1] + -15.308;
   1:  PR[91,2] = PR[90,2] + 1.427;
   1:L PR[91] R[100]mm/sec CNT100;
   1:  PR[91,1] = PR[90,1] + -21.414;
   1:  PR[91,2] = PR[90,2] + -4.679;
   1:L PR[91] R[100]mm/sec CNT100;
   1:  PR[92] = PR[91];
   1:  PR[92,3] = PR[92,3] + R[101];
   1:J PR[92] R[102]% CNT100;
   1:  PR[91,1] = PR[90,1] + 45.809;
   1:  PR[91,2] = PR[90,2] + 28.025;
   1:  PR[92] = PR[91];
   1:  PR[92,3] = PR[92,3] + R[101];
   1:J PR[92] R[102]% CNT100;
   1:L PR[91] 100mm/sec CNT100 RampTo R[100];
   1:  PR[91,1] = PR[90,1] + 45.333;
   1:  PR[91,2] = PR[90,2] + 28.527;
   1:L PR[91] R[100]mm/sec CNT100;
   1:  PR[91,1] = PR[90,1] + 45.004;
   1:  PR[91,2] = PR[90,2] + 28.696;
   1:L PR[91] R[100]mm/sec CNT100;
   1:  PR[91,1] = PR[90,1] + 44.632;
   1:  PR[91,2] = PR[90,2] + 28.827;
   1:L PR[91] R[100]mm/sec CNT100;
   1:  PR[91,1] = PR[90,1] + 44.400;
   1:  PR[91,2] = PR[90,2] + 28.866;
   1:L PR[91] R[100]mm/sec CNT100;
   1:  PR[91,1] = PR[90,1] + 43.686;
   1:  PR[91,2] = PR[90,2] + 29.176;
   1:L PR[91] R[100]mm/sec CNT100;
   1:  PR[91,1] = PR[90,1] + 43.606;
   1:  PR[91,2] = PR[90,2] + 29.232;
   1:L PR[91] R[100]mm/sec CNT100;
   1:  PR[91,1] = PR[90,1] + 43.130;
   1:  PR[91,2] = PR[90,2] + 29.340;
   1:L PR[91] R[100]mm/sec CNT100;
   1:  PR[91,1] = PR[90,1] + 42.970;
   1:  PR[91,2] = PR[90,2] + 29.348;
   1:L PR[91] R[100]mm/sec CNT100;
   1:  PR[91,1] = PR[90,1] + 42.159;
   1:  PR[91,2] = PR[90,2] + 29.341;
   1:L PR[91] R[100]mm/sec CNT100;
   1:  PR[91,1] = PR[90,1] + 41.389;
   1:  PR[91,2] = PR[90,2] + 29.176;
   1:L PR[91] R[100]mm/sec CNT100;
   1:  PR[91,1] = PR[90,1] + 41.264;
   1:  PR[91,2] = PR[90,2] + 29.115;
   1:L PR[91] R[100]mm/sec CNT100;
   1:  PR[91,1] = PR[90,1] + 40.574;
   1:  PR[91,2] = PR[90,2] + 28.853;
   1:L PR[91] R[100]mm/sec CNT100;
   1:  PR[91,1] = PR[90,1] + 40.084;
   1:  PR[91,2] = PR[90,2] + 28.620;
   1:L PR[91] R[100]mm/sec CNT100;
   1:  PR[91,1] = PR[90,1] + 39.744;
   1:  PR[91,2] = PR[90,2] + 28.488;
   1:L PR[91] R[100]mm/sec CNT100;
   1:  PR[91,1] = PR[90,1] + 38.989;
   1:  PR[91,2] = PR[90,2] + 27.866;
   1:L PR[91] R[100]mm/sec CNT100;
   1:  PR[91,1] = PR[90,1] + 38.628;
   1:  PR[91,2] = PR[90,2] + 27.497;
   1:L PR[91] R[100]mm/sec CNT100;
   1:  PR[91,1] = PR[90,1] + 38.093;
   1:  PR[91,2] = PR[90,2] + 26.770;
   1:L PR[91] R[100]mm/sec CNT100;
   1:  PR[91,1] = PR[90,1] + 38.025;
   1:  PR[91,2] = PR[90,2] + 26.556;
   1:L PR[91] R[100]mm/sec CNT100;
   1:  PR[91,1] = PR[90,1] + 37.706;
   1:  PR[91,2] = PR[90,2] + 25.910;
   1:L PR[91] R[100]mm/sec CNT100;
   1:  PR[91,1] = PR[90,1] + 37.497;
   1:  PR[91,2] = PR[90,2] + 25.156;
   1:L PR[91] R[100]mm/sec CNT100;
   1:  PR[91,1] = PR[90,1] + 37.299;
   1:  PR[91,2] = PR[90,2] + 24.230;
   1:L PR[91] R[100]mm/sec CNT100;
   1:  PR[91,1] = PR[90,1] + 37.258;
   1:  PR[91,2] = PR[90,2] + 23.374;
   1:L PR[91] R[100]mm/sec CNT100;
   1:  PR[91,1] = PR[90,1] + 37.255;
   1:  PR[91,2] = PR[90,2] + 22.399;
   1:L PR[91] R[100]mm/sec CNT100;
   1:  PR[91,1] = PR[90,1] + 37.256;
   1:  PR[91,2] = PR[90,2] + 3.183;
   1:L PR[91] R[100]mm/sec CNT100;
   1:  PR[91,1] = PR[90,1] + 37.263;
   1:  PR[91,2] = PR[90,2] + 1.992;
   1:L PR[91] R[100]mm/sec CNT100;
   1:  PR[91,1] = PR[90,1] + 37.284;
   1:  PR[91,2] = PR[90,2] + 1.232;
   1:L PR[91] R[100]mm/sec CNT100;
   1:  PR[91,1] = PR[90,1] + 37.361;
   1:  PR[91,2] = PR[90,2] + 0.213;
   1:L PR[91] R[100]mm/sec CNT100;
   1:  PR[91,1] = PR[90,1] + 37.483;
   1:  PR[91,2] = PR[90,2] + -0.635;
   1:L PR[91] R[100]mm/sec CNT100;
   1:  PR[91,1] = PR[90,1] + 37.638;
   1:  PR[91,2] = PR[90,2] + -1.544;
   1:L PR[91] R[100]mm/sec CNT100;
   1:  PR[91,1] = PR[90,1] + 37.644;
   1:  PR[91,2] = PR[90,2] + -1.720;
   1:L PR[91] R[100]mm/sec CNT100;
   1:  PR[91,1] = PR[90,1] + 37.764;
   1:  PR[91,2] = PR[90,2] + -2.402;
   1:L PR[91] R[100]mm/sec CNT100;
   1:  PR[91,1] = PR[90,1] + 37.786;
   1:  PR[91,2] = PR[90,2] + -2.749;
   1:L PR[91] R[100]mm/sec CNT100;
   1:  PR[91,1] = PR[90,1] + 37.853;
   1:  PR[91,2] = PR[90,2] + -3.268;
   1:L PR[91] R[100]mm/sec CNT100;
   1:  PR[91,1] = PR[90,1] + 37.927;
   1:  PR[91,2] = PR[90,2] + -3.691;
   1:L PR[91] R[100]mm/sec CNT100;
   1:  PR[91,1] = PR[90,1] + 37.969;
   1:  PR[91,2] = PR[90,2] + -4.078;
   1:L PR[91] R[100]mm/sec CNT100;
   1:  PR[91,1] = PR[90,1] + 38.128;
   1:  PR[91,2] = PR[90,2] + -4.599;
   1:L PR[91] R[100]mm/sec CNT100;
   1:  PR[91,1] = PR[90,1] + 38.149;
   1:  PR[91,2] = PR[90,2] + -4.764;
   1:L PR[91] R[100]mm/sec CNT100;
   1:  PR[91,1] = PR[90,1] + 38.312;
   1:  PR[91,2] = PR[90,2] + -5.105;
   1:L PR[91] R[100]mm/sec CNT100;
   1:  PR[91,1] = PR[90,1] + 38.487;
   1:  PR[91,2] = PR[90,2] + -5.445;
   1:L PR[91] R[100]mm/sec CNT100;
   1:  PR[91,1] = PR[90,1] + 38.500;
   1:  PR[91,2] = PR[90,2] + -5.585;
   1:L PR[91] R[100]mm/sec CNT100;
   1:  PR[91,1] = PR[90,1] + 38.748;
   1:  PR[91,2] = PR[90,2] + -6.241;
   1:L PR[91] R[100]mm/sec CNT100;
   1:  PR[91,1] = PR[90,1] + 38.810;
   1:  PR[91,2] = PR[90,2] + -6.678;
   1:L PR[91] R[100]mm/sec CNT100;
   1:  PR[91,1] = PR[90,1] + 38.887;
   1:  PR[91,2] = PR[90,2] + -7.044;
   1:L PR[91] R[100]mm/sec CNT100;
   1:  PR[91,1] = PR[90,1] + 39.084;
   1:  PR[91,2] = PR[90,2] + -7.552;
   1:L PR[91] R[100]mm/sec CNT100;
   1:  PR[91,1] = PR[90,1] + 39.096;
   1:  PR[91,2] = PR[90,2] + -7.627;
   1:L PR[91] R[100]mm/sec CNT100;
   1:  PR[91,1] = PR[90,1] + 39.552;
   1:  PR[91,2] = PR[90,2] + -8.214;
   1:L PR[91] R[100]mm/sec CNT100;
   1:  PR[91,1] = PR[90,1] + 39.601;
   1:  PR[91,2] = PR[90,2] + -8.582;
   1:L PR[91] R[100]mm/sec CNT100;
   1:  PR[91,1] = PR[90,1] + 39.785;
   1:  PR[91,2] = PR[90,2] + -9.050;
   1:L PR[91] R[100]mm/sec CNT100;
   1:  PR[91,1] = PR[90,1] + 39.963;
   1:  PR[91,2] = PR[90,2] + -9.570;
   1:L PR[91] R[100]mm/sec CNT100;
   1:  PR[91,1] = PR[90,1] + 39.985;
   1:  PR[91,2] = PR[90,2] + -9.670;
   1:L PR[91] R[100]mm/sec CNT100;
   1:  PR[91,1] = PR[90,1] + 40.053;
   1:  PR[91,2] = PR[90,2] + -9.750;
   1:L PR[91] R[100]mm/sec CNT100;
   1:  PR[91,1] = PR[90,1] + 40.466;
   1:  PR[91,2] = PR[90,2] + -10.117;
   1:L PR[91] R[100]mm/sec CNT100;
   1:  PR[91,1] = PR[90,1] + 40.533;
   1:  PR[91,2] = PR[90,2] + -10.516;
   1:L PR[91] R[100]mm/sec CNT100;
   1:  PR[91,1] = PR[90,1] + 40.747;
   1:  PR[91,2] = PR[90,2] + -10.945;
   1:L PR[91] R[100]mm/sec CNT100;
   1:  PR[91,1] = PR[90,1] + 40.987;
   1:  PR[91,2] = PR[90,2] + -11.490;
   1:L PR[91] R[100]mm/sec CNT100;
   1:  PR[91,1] = PR[90,1] + 41.544;
   1:  PR[91,2] = PR[90,2] + -11.958;
   1:L PR[91] R[100]mm/sec CNT100;
   1:  PR[91,1] = PR[90,1] + 41.682;
   1:  PR[91,2] = PR[90,2] + -12.529;
   1:L PR[91] R[100]mm/sec CNT100;
   1:  PR[91,1] = PR[90,1] + 41.772;
   1:  PR[91,2] = PR[90,2] + -12.737;
   1:L PR[91] R[100]mm/sec CNT100;
   1:  PR[91,1] = PR[90,1] + 42.270;
   1:  PR[91,2] = PR[90,2] + -13.353;
   1:L PR[91] R[100]mm/sec CNT100;
   1:  PR[91,1] = PR[90,1] + 42.629;
   1:  PR[91,2] = PR[90,2] + -13.798;
   1:L PR[91] R[100]mm/sec CNT100;
   1:  PR[91,1] = PR[90,1] + 42.920;
   1:  PR[91,2] = PR[90,2] + -14.327;
   1:L PR[91] R[100]mm/sec CNT100;
   1:  PR[91,1] = PR[90,1] + 43.518;
   1:  PR[91,2] = PR[90,2] + -14.774;
   1:L PR[91] R[100]mm/sec CNT100;
   1:  PR[91,1] = PR[90,1] + 43.792;
   1:  PR[91,2] = PR[90,2] + -15.410;
   1:L PR[91] R[100]mm/sec CNT100;
   1:  PR[91,1] = PR[90,1] + 44.418;
   1:  PR[91,2] = PR[90,2] + -15.747;
   1:L PR[91] R[100]mm/sec CNT100;
   1:  PR[91,1] = PR[90,1] + 44.693;
   1:  PR[91,2] = PR[90,2] + -16.411;
   1:L PR[91] R[100]mm/sec CNT100;
   1:  PR[91,1] = PR[90,1] + 44.699;
   1:  PR[91,2] = PR[90,2] + -16.422;
   1:L PR[91] R[100]mm/sec CNT100;
   1:  PR[91,1] = PR[90,1] + 44.704;
   1:  PR[91,2] = PR[90,2] + -16.426;
   1:L PR[91] R[100]mm/sec CNT100;
   1:  PR[91,1] = PR[90,1] + 45.349;
   1:  PR[91,2] = PR[90,2] + -16.715;
   1:L PR[91] R[100]mm/sec CNT100;
   1:  PR[91,1] = PR[90,1] + 45.643;
   1:  PR[91,2] = PR[90,2] + -17.365;
   1:L PR[91] R[100]mm/sec CNT100;
   1:  PR[91,1] = PR[90,1] + 45.648;
   1:  PR[91,2] = PR[90,2] + -17.372;
   1:L PR[91] R[100]mm/sec CNT100;
   1:  PR[91,1] = PR[90,1] + 45.658;
   1:  PR[91,2] = PR[90,2] + -17.377;
   1:L PR[91] R[100]mm/sec CNT100;
   1:  PR[91,1] = PR[90,1] + 46.291;
   1:  PR[91,2] = PR[90,2] + -17.646;
   1:L PR[91] R[100]mm/sec CNT100;
   1:  PR[91,1] = PR[90,1] + 46.674;
   1:  PR[91,2] = PR[90,2] + -18.294;
   1:L PR[91] R[100]mm/sec CNT100;
   1:  PR[91,1] = PR[90,1] + 47.261;
   1:  PR[91,2] = PR[90,2] + -18.556;
   1:L PR[91] R[100]mm/sec CNT100;
   1:  PR[91,1] = PR[90,1] + 47.742;
   1:  PR[91,2] = PR[90,2] + -19.150;
   1:L PR[91] R[100]mm/sec CNT100;
   1:  PR[91,1] = PR[90,1] + 48.248;
   1:  PR[91,2] = PR[90,2] + -19.458;
   1:L PR[91] R[100]mm/sec CNT100;
   1:  PR[91,1] = PR[90,1] + 48.672;
   1:  PR[91,2] = PR[90,2] + -19.769;
   1:L PR[91] R[100]mm/sec CNT100;
   1:  PR[91,1] = PR[90,1] + 48.728;
   1:  PR[91,2] = PR[90,2] + -19.782;
   1:L PR[91] R[100]mm/sec CNT100;
   1:  PR[91,1] = PR[90,1] + 48.929;
   1:  PR[91,2] = PR[90,2] + -19.959;
   1:L PR[91] R[100]mm/sec CNT100;
   1:  PR[91,1] = PR[90,1] + 49.113;
   1:  PR[91,2] = PR[90,2] + -20.094;
   1:L PR[91] R[100]mm/sec CNT100;
   1:  PR[91,1] = PR[90,1] + 49.139;
   1:  PR[91,2] = PR[90,2] + -20.143;
   1:L PR[91] R[100]mm/sec CNT100;
   1:  PR[91,1] = PR[90,1] + 49.330;
   1:  PR[91,2] = PR[90,2] + -20.310;
   1:L PR[91] R[100]mm/sec CNT100;
   1:  PR[91,1] = PR[90,1] + 49.509;
   1:  PR[91,2] = PR[90,2] + -20.383;
   1:L PR[91] R[100]mm/sec CNT100;
   1:  PR[91,1] = PR[90,1] + 50.060;
   1:  PR[91,2] = PR[90,2] + -20.532;
   1:L PR[91] R[100]mm/sec CNT100;
   1:  PR[91,1] = PR[90,1] + 50.591;
   1:  PR[91,2] = PR[90,2] + -21.083;
   1:L PR[91] R[100]mm/sec CNT100;
   1:  PR[91,1] = PR[90,1] + 51.100;
   1:  PR[91,2] = PR[90,2] + -21.345;
   1:L PR[91] R[100]mm/sec CNT100;
   1:  PR[91,1] = PR[90,1] + 51.480;
   1:  PR[91,2] = PR[90,2] + -21.511;
   1:L PR[91] R[100]mm/sec CNT100;
   1:  PR[91,1] = PR[90,1] + 51.881;
   1:  PR[91,2] = PR[90,2] + -21.584;
   1:L PR[91] R[100]mm/sec CNT100;
   1:  PR[91,1] = PR[90,1] + 52.426;
   1:  PR[91,2] = PR[90,2] + -22.091;
   1:L PR[91] R[100]mm/sec CNT100;
   1:  PR[91,1] = PR[90,1] + 52.492;
   1:  PR[91,2] = PR[90,2] + -22.106;
   1:L PR[91] R[100]mm/sec CNT100;
   1:  PR[91,1] = PR[90,1] + 52.989;
   1:  PR[91,2] = PR[90,2] + -22.308;
   1:L PR[91] R[100]mm/sec CNT100;
   1:  PR[91,1] = PR[90,1] + 53.408;
   1:  PR[91,2] = PR[90,2] + -22.451;
   1:L PR[91] R[100]mm/sec CNT100;
   1:  PR[91,1] = PR[90,1] + 53.797;
   1:  PR[91,2] = PR[90,2] + -22.511;
   1:L PR[91] R[100]mm/sec CNT100;
   1:  PR[91,1] = PR[90,1] + 54.422;
   1:  PR[91,2] = PR[90,2] + -22.928;
   1:L PR[91] R[100]mm/sec CNT100;
   1:  PR[91,1] = PR[90,1] + 54.462;
   1:  PR[91,2] = PR[90,2] + -22.960;
   1:L PR[91] R[100]mm/sec CNT100;
   1:  PR[91,1] = PR[90,1] + 54.496;
   1:  PR[91,2] = PR[90,2] + -22.966;
   1:L PR[91] R[100]mm/sec CNT100;
   1:  PR[91,1] = PR[90,1] + 55.008;
   1:  PR[91,2] = PR[90,2] + -23.197;
   1:L PR[91] R[100]mm/sec CNT100;
   1:  PR[91,1] = PR[90,1] + 55.768;
   1:  PR[91,2] = PR[90,2] + -23.336;
   1:L PR[91] R[100]mm/sec CNT100;
   1:  PR[91,1] = PR[90,1] + 56.365;
   1:  PR[91,2] = PR[90,2] + -23.522;
   1:L PR[91] R[100]mm/sec CNT100;
   1:  PR[91,1] = PR[90,1] + 56.586;
   1:  PR[91,2] = PR[90,2] + -23.545;
   1:L PR[91] R[100]mm/sec CNT100;
   1:  PR[91,1] = PR[90,1] + 57.156;
   1:  PR[91,2] = PR[90,2] + -23.797;
   1:L PR[91] R[100]mm/sec CNT100;
   1:  PR[91,1] = PR[90,1] + 57.335;
   1:  PR[91,2] = PR[90,2] + -23.892;
   1:L PR[91] R[100]mm/sec CNT100;
   1:  PR[91,1] = PR[90,1] + 57.413;
   1:  PR[91,2] = PR[90,2] + -23.902;
   1:L PR[91] R[100]mm/sec CNT100;
   1:  PR[91,1] = PR[90,1] + 57.977;
   1:  PR[91,2] = PR[90,2] + -24.096;
   1:L PR[91] R[100]mm/sec CNT100;
   1:  PR[91,1] = PR[90,1] + 58.307;
   1:  PR[91,2] = PR[90,2] + -24.130;
   1:L PR[91] R[100]mm/sec CNT100;
   1:  PR[91,1] = PR[90,1] + 58.751;
   1:  PR[91,2] = PR[90,2] + -24.225;
   1:L PR[91] R[100]mm/sec CNT100;
   1:  PR[91,1] = PR[90,1] + 59.610;
   1:  PR[91,2] = PR[90,2] + -24.307;
   1:L PR[91] R[100]mm/sec CNT100;
   1:  PR[91,1] = PR[90,1] + 60.215;
   1:  PR[91,2] = PR[90,2] + -24.389;
   1:L PR[91] R[100]mm/sec CNT100;
   1:  PR[91,1] = PR[90,1] + 60.489;
   1:  PR[91,2] = PR[90,2] + -24.400;
   1:L PR[91] R[100]mm/sec CNT100;
   1:  PR[91,1] = PR[90,1] + 61.223;
   1:  PR[91,2] = PR[90,2] + -24.510;
   1:L PR[91] R[100]mm/sec CNT100;
   1:  PR[91,1] = PR[90,1] + 61.346;
   1:  PR[91,2] = PR[90,2] + -24.514;
   1:L PR[91] R[100]mm/sec CNT100;
   1:  PR[91,1] = PR[90,1] + 62.239;
   1:  PR[91,2] = PR[90,2] + -24.619;
   1:L PR[91] R[100]mm/sec CNT100;
   1:  PR[91,1] = PR[90,1] + 63.151;
   1:  PR[91,2] = PR[90,2] + -24.690;
   1:L PR[91] R[100]mm/sec CNT100;
   1:  PR[91,1] = PR[90,1] + 64.103;
   1:  PR[91,2] = PR[90,2] + -24.718;
   1:L PR[91] R[100]mm/sec CNT100;
   1:  PR[91,1] = PR[90,1] + 65.029;
   1:  PR[91,2] = PR[90,2] + -24.690;
   1:L PR[91] R[100]mm/sec CNT100;
   1:  PR[91,1] = PR[90,1] + 66.035;
   1:  PR[91,2] = PR[90,2] + -24.612;
   1:L PR[91] R[100]mm/sec CNT100;
   1:  PR[91,1] = PR[90,1] + 67.116;
   1:  PR[91,2] = PR[90,2] + -24.506;
   1:L PR[91] R[100]mm/sec CNT100;
   1:  PR[91,1] = PR[90,1] + 68.890;
   1:  PR[91,2] = PR[90,2] + -24.290;
   1:L PR[91] R[100]mm/sec CNT100;
   1:  PR[91,1] = PR[90,1] + 69.388;
   1:  PR[91,2] = PR[90,2] + -24.189;
   1:L PR[91] R[100]mm/sec CNT100;
   1:  PR[91,1] = PR[90,1] + 69.849;
   1:  PR[91,2] = PR[90,2] + -24.143;
   1:L PR[91] R[100]mm/sec CNT100;
   1:  PR[91,1] = PR[90,1] + 70.580;
   1:  PR[91,2] = PR[90,2] + -23.932;
   1:L PR[91] R[100]mm/sec CNT100;
   1:  PR[91,1] = PR[90,1] + 70.761;
   1:  PR[91,2] = PR[90,2] + -23.909;
   1:L PR[91] R[100]mm/sec CNT100;
   1:  PR[91,1] = PR[90,1] + 71.186;
   1:  PR[91,2] = PR[90,2] + -23.739;
   1:L PR[91] R[100]mm/sec CNT100;
   1:  PR[91,1] = PR[90,1] + 71.720;
   1:  PR[91,2] = PR[90,2] + -23.561;
   1:L PR[91] R[100]mm/sec CNT100;
   1:  PR[91,1] = PR[90,1] + 72.690;
   1:  PR[91,2] = PR[90,2] + -23.312;
   1:L PR[91] R[100]mm/sec CNT100;
   1:  PR[91,1] = PR[90,1] + 73.371;
   1:  PR[91,2] = PR[90,2] + -23.049;
   1:L PR[91] R[100]mm/sec CNT100;
   1:  PR[91,1] = PR[90,1] + 73.631;
   1:  PR[91,2] = PR[90,2] + -22.992;
   1:L PR[91] R[100]mm/sec CNT100;
   1:  PR[91,1] = PR[90,1] + 74.013;
   1:  PR[91,2] = PR[90,2] + -22.788;
   1:L PR[91] R[100]mm/sec CNT100;
   1:  PR[91,1] = PR[90,1] + 74.574;
   1:  PR[91,2] = PR[90,2] + -22.538;
   1:L PR[91] R[100]mm/sec CNT100;
   1:  PR[91,1] = PR[90,1] + 74.992;
   1:  PR[91,2] = PR[90,2] + -22.370;
   1:L PR[91] R[100]mm/sec CNT100;
   1:  PR[91,1] = PR[90,1] + 75.534;
   1:  PR[91,2] = PR[90,2] + -22.183;
   1:L PR[91] R[100]mm/sec CNT100;
   1:  PR[91,1] = PR[90,1] + 76.473;
   1:  PR[91,2] = PR[90,2] + -21.633;
   1:L PR[91] R[100]mm/sec CNT100;
   1:  PR[91,1] = PR[90,1] + 77.422;
   1:  PR[91,2] = PR[90,2] + -21.192;
   1:L PR[91] R[100]mm/sec CNT100;
   1:  PR[91,1] = PR[90,1] + 77.879;
   1:  PR[91,2] = PR[90,2] + -20.872;
   1:L PR[91] R[100]mm/sec CNT100;
   1:  PR[91,1] = PR[90,1] + 79.277;
   1:  PR[91,2] = PR[90,2] + -19.951;
   1:L PR[91] R[100]mm/sec CNT100;
   1:  PR[91,1] = PR[90,1] + 79.407;
   1:  PR[91,2] = PR[90,2] + -19.882;
   1:L PR[91] R[100]mm/sec CNT100;
   1:  PR[91,1] = PR[90,1] + 80.286;
   1:  PR[91,2] = PR[90,2] + -19.283;
   1:L PR[91] R[100]mm/sec CNT100;
   1:  PR[91,1] = PR[90,1] + 81.212;
   1:  PR[91,2] = PR[90,2] + -18.514;
   1:L PR[91] R[100]mm/sec CNT100;
   1:  PR[91,1] = PR[90,1] + 82.174;
   1:  PR[91,2] = PR[90,2] + -17.646;
   1:L PR[91] R[100]mm/sec CNT100;
   1:  PR[91,1] = PR[90,1] + 83.136;
   1:  PR[91,2] = PR[90,2] + -16.710;
   1:L PR[91] R[100]mm/sec CNT100;
   1:  PR[91,1] = PR[90,1] + 84.102;
   1:  PR[91,2] = PR[90,2] + -15.688;
   1:L PR[91] R[100]mm/sec CNT100;
   1:  PR[91,1] = PR[90,1] + 84.651;
   1:  PR[91,2] = PR[90,2] + -15.067;
   1:L PR[91] R[100]mm/sec CNT100;
   1:  PR[91,1] = PR[90,1] + 85.435;
   1:  PR[91,2] = PR[90,2] + -14.122;
   1:L PR[91] R[100]mm/sec CNT100;
   1:  PR[91,1] = PR[90,1] + 86.023;
   1:  PR[91,2] = PR[90,2] + -13.280;
   1:L PR[91] R[100]mm/sec CNT100;
   1:  PR[91,1] = PR[90,1] + 86.103;
   1:  PR[91,2] = PR[90,2] + -13.182;
   1:L PR[91] R[100]mm/sec CNT100;
   1:  PR[91,1] = PR[90,1] + 86.219;
   1:  PR[91,2] = PR[90,2] + -12.965;
   1:L PR[91] R[100]mm/sec CNT100;
   1:  PR[91,1] = PR[90,1] + 86.713;
   1:  PR[91,2] = PR[90,2] + -12.186;
   1:L PR[91] R[100]mm/sec CNT100;
   1:  PR[91,1] = PR[90,1] + 87.350;
   1:  PR[91,2] = PR[90,2] + -11.244;
   1:L PR[91] R[100]mm/sec CNT100;
   1:  PR[91,1] = PR[90,1] + 87.813;
   1:  PR[91,2] = PR[90,2] + -10.292;
   1:L PR[91] R[100]mm/sec CNT100;
   1:  PR[91,1] = PR[90,1] + 88.344;
   1:  PR[91,2] = PR[90,2] + -9.337;
   1:L PR[91] R[100]mm/sec CNT100;
   1:  PR[91,1] = PR[90,1] + 88.720;
   1:  PR[91,2] = PR[90,2] + -8.355;
   1:L PR[91] R[100]mm/sec CNT100;
   1:  PR[91,1] = PR[90,1] + 89.178;
   1:  PR[91,2] = PR[90,2] + -7.441;
   1:L PR[91] R[100]mm/sec CNT100;
   1:  PR[91,1] = PR[90,1] + 89.260;
   1:  PR[91,2] = PR[90,2] + -7.077;
   1:L PR[91] R[100]mm/sec CNT100;
   1:  PR[91,1] = PR[90,1] + 89.454;
   1:  PR[91,2] = PR[90,2] + -6.473;
   1:L PR[91] R[100]mm/sec CNT100;
   1:  PR[91,1] = PR[90,1] + 89.797;
   1:  PR[91,2] = PR[90,2] + -5.435;
   1:L PR[91] R[100]mm/sec CNT100;
   1:  PR[91,1] = PR[90,1] + 90.107;
   1:  PR[91,2] = PR[90,2] + -4.580;
   1:L PR[91] R[100]mm/sec CNT100;
   1:  PR[91,1] = PR[90,1] + 90.137;
   1:  PR[91,2] = PR[90,2] + -4.281;
   1:L PR[91] R[100]mm/sec CNT100;
   1:  PR[91,1] = PR[90,1] + 90.298;
   1:  PR[91,2] = PR[90,2] + -3.616;
   1:L PR[91] R[100]mm/sec CNT100;
   1:  PR[91,1] = PR[90,1] + 90.440;
   1:  PR[91,2] = PR[90,2] + -2.653;
   1:L PR[91] R[100]mm/sec CNT100;
   1:  PR[91,1] = PR[90,1] + 90.577;
   1:  PR[91,2] = PR[90,2] + -1.868;
   1:L PR[91] R[100]mm/sec CNT100;
   1:  PR[91,1] = PR[90,1] + 90.590;
   1:  PR[91,2] = PR[90,2] + -1.706;
   1:L PR[91] R[100]mm/sec CNT100;
   1:  PR[91,1] = PR[90,1] + 90.894;
   1:  PR[91,2] = PR[90,2] + 0.314;
   1:L PR[91] R[100]mm/sec CNT100;
   1:  PR[91,1] = PR[90,1] + 90.966;
   1:  PR[91,2] = PR[90,2] + 1.240;
   1:L PR[91] R[100]mm/sec CNT100;
   1:  PR[91,1] = PR[90,1] + 91.000;
   1:  PR[91,2] = PR[90,2] + 2.194;
   1:L PR[91] R[100]mm/sec CNT100;
   1:  PR[91,1] = PR[90,1] + 91.008;
   1:  PR[91,2] = PR[90,2] + 22.396;
   1:L PR[91] R[100]mm/sec CNT100;
   1:  PR[91,1] = PR[90,1] + 90.998;
   1:  PR[91,2] = PR[90,2] + 23.615;
   1:L PR[91] R[100]mm/sec CNT100;
   1:  PR[91,1] = PR[90,1] + 90.952;
   1:  PR[91,2] = PR[90,2] + 24.355;
   1:L PR[91] R[100]mm/sec CNT100;
   1:  PR[91,1] = PR[90,1] + 90.788;
   1:  PR[91,2] = PR[90,2] + 24.903;
   1:L PR[91] R[100]mm/sec CNT100;
   1:  PR[91,1] = PR[90,1] + 90.760;
   1:  PR[91,2] = PR[90,2] + 25.043;
   1:L PR[91] R[100]mm/sec CNT100;
   1:  PR[91,1] = PR[90,1] + 90.514;
   1:  PR[91,2] = PR[90,2] + 25.765;
   1:L PR[91] R[100]mm/sec CNT100;
   1:  PR[91,1] = PR[90,1] + 90.377;
   1:  PR[91,2] = PR[90,2] + 26.409;
   1:L PR[91] R[100]mm/sec CNT100;
   1:  PR[91,1] = PR[90,1] + 90.249;
   1:  PR[91,2] = PR[90,2] + 26.603;
   1:L PR[91] R[100]mm/sec CNT100;
   1:  PR[91,1] = PR[90,1] + 89.703;
   1:  PR[91,2] = PR[90,2] + 27.283;
   1:L PR[91] R[100]mm/sec CNT100;
   1:  PR[91,1] = PR[90,1] + 89.435;
   1:  PR[91,2] = PR[90,2] + 27.709;
   1:L PR[91] R[100]mm/sec CNT100;
   1:  PR[91,1] = PR[90,1] + 88.984;
   1:  PR[91,2] = PR[90,2] + 28.006;
   1:L PR[91] R[100]mm/sec CNT100;
   1:  PR[91,1] = PR[90,1] + 88.472;
   1:  PR[91,2] = PR[90,2] + 28.510;
   1:L PR[91] R[100]mm/sec CNT100;
   1:  PR[91,1] = PR[90,1] + 88.177;
   1:  PR[91,2] = PR[90,2] + 28.684;
   1:L PR[91] R[100]mm/sec CNT100;
   1:  PR[91,1] = PR[90,1] + 87.856;
   1:  PR[91,2] = PR[90,2] + 28.788;
   1:L PR[91] R[100]mm/sec CNT100;
   1:  PR[91,1] = PR[90,1] + 87.573;
   1:  PR[91,2] = PR[90,2] + 28.840;
   1:L PR[91] R[100]mm/sec CNT100;
   1:  PR[91,1] = PR[90,1] + 86.769;
   1:  PR[91,2] = PR[90,2] + 29.193;
   1:L PR[91] R[100]mm/sec CNT100;
   1:  PR[91,1] = PR[90,1] + 86.730;
   1:  PR[91,2] = PR[90,2] + 29.223;
   1:L PR[91] R[100]mm/sec CNT100;
   1:  PR[91,1] = PR[90,1] + 86.309;
   1:  PR[91,2] = PR[90,2] + 29.333;
   1:L PR[91] R[100]mm/sec CNT100;
   1:  PR[91,1] = PR[90,1] + 86.170;
   1:  PR[91,2] = PR[90,2] + 29.340;
   1:L PR[91] R[100]mm/sec CNT100;
   1:  PR[91,1] = PR[90,1] + 85.347;
   1:  PR[91,2] = PR[90,2] + 29.345;
   1:L PR[91] R[100]mm/sec CNT100;
   1:  PR[91,1] = PR[90,1] + 84.585;
   1:  PR[91,2] = PR[90,2] + 29.199;
   1:L PR[91] R[100]mm/sec CNT100;
   1:  PR[91,1] = PR[90,1] + 84.568;
   1:  PR[91,2] = PR[90,2] + 29.198;
   1:L PR[91] R[100]mm/sec CNT100;
   1:  PR[91,1] = PR[90,1] + 84.364;
   1:  PR[91,2] = PR[90,2] + 29.106;
   1:L PR[91] R[100]mm/sec CNT100;
   1:  PR[91,1] = PR[90,1] + 83.766;
   1:  PR[91,2] = PR[90,2] + 28.884;
   1:L PR[91] R[100]mm/sec CNT100;
   1:  PR[91,1] = PR[90,1] + 83.386;
   1:  PR[91,2] = PR[90,2] + 28.715;
   1:L PR[91] R[100]mm/sec CNT100;
   1:  PR[91,1] = PR[90,1] + 82.954;
   1:  PR[91,2] = PR[90,2] + 28.546;
   1:L PR[91] R[100]mm/sec CNT100;
   1:  PR[91,1] = PR[90,1] + 82.196;
   1:  PR[91,2] = PR[90,2] + 27.938;
   1:L PR[91] R[100]mm/sec CNT100;
   1:  PR[91,1] = PR[90,1] + 81.749;
   1:  PR[91,2] = PR[90,2] + 27.485;
   1:L PR[91] R[100]mm/sec CNT100;
   1:  PR[91,1] = PR[90,1] + 81.179;
   1:  PR[91,2] = PR[90,2] + 26.739;
   1:L PR[91] R[100]mm/sec CNT100;
   1:  PR[91,1] = PR[90,1] + 81.048;
   1:  PR[91,2] = PR[90,2] + 26.362;
   1:L PR[91] R[100]mm/sec CNT100;
   1:  PR[91,1] = PR[90,1] + 80.834;
   1:  PR[91,2] = PR[90,2] + 25.905;
   1:L PR[91] R[100]mm/sec CNT100;
   1:  PR[91,1] = PR[90,1] + 80.589;
   1:  PR[91,2] = PR[90,2] + 25.117;
   1:L PR[91] R[100]mm/sec CNT100;
   1:  PR[91,1] = PR[90,1] + 80.557;
   1:  PR[91,2] = PR[90,2] + 25.041;
   1:L PR[91] R[100]mm/sec CNT100;
   1:  PR[91,1] = PR[90,1] + 80.386;
   1:  PR[91,2] = PR[90,2] + 24.233;
   1:L PR[91] R[100]mm/sec CNT100;
   1:  PR[91,1] = PR[90,1] + 80.347;
   1:  PR[91,2] = PR[90,2] + 23.375;
   1:L PR[91] R[100]mm/sec CNT100;
   1:  PR[91,1] = PR[90,1] + 80.342;
   1:  PR[91,2] = PR[90,2] + 22.398;
   1:L PR[91] R[100]mm/sec CNT100;
   1:  PR[91,1] = PR[90,1] + 80.340;
   1:  PR[91,2] = PR[90,2] + 3.168;
   1:L PR[91] R[100]mm/sec CNT100;
   1:  PR[91,1] = PR[90,1] + 80.319;
   1:  PR[91,2] = PR[90,2] + 1.749;
   1:L PR[91] R[100]mm/sec CNT100;
   1:  PR[91,1] = PR[90,1] + 80.249;
   1:  PR[91,2] = PR[90,2] + 0.599;
   1:L PR[91] R[100]mm/sec CNT100;
   1:  PR[91,1] = PR[90,1] + 80.111;
   1:  PR[91,2] = PR[90,2] + -0.635;
   1:L PR[91] R[100]mm/sec CNT100;
   1:  PR[91,1] = PR[90,1] + 79.800;
   1:  PR[91,2] = PR[90,2] + -2.279;
   1:L PR[91] R[100]mm/sec CNT100;
   1:  PR[91,1] = PR[90,1] + 79.559;
   1:  PR[91,2] = PR[90,2] + -2.940;
   1:L PR[91] R[100]mm/sec CNT100;
   1:  PR[91,1] = PR[90,1] + 79.329;
   1:  PR[91,2] = PR[90,2] + -3.422;
   1:L PR[91] R[100]mm/sec CNT100;
   1:  PR[91,1] = PR[90,1] + 79.233;
   1:  PR[91,2] = PR[90,2] + -3.763;
   1:L PR[91] R[100]mm/sec CNT100;
   1:  PR[91,1] = PR[90,1] + 78.487;
   1:  PR[91,2] = PR[90,2] + -5.420;
   1:L PR[91] R[100]mm/sec CNT100;
   1:  PR[91,1] = PR[90,1] + 78.328;
   1:  PR[91,2] = PR[90,2] + -5.661;
   1:L PR[91] R[100]mm/sec CNT100;
   1:  PR[91,1] = PR[90,1] + 78.197;
   1:  PR[91,2] = PR[90,2] + -5.929;
   1:L PR[91] R[100]mm/sec CNT100;
   1:  PR[91,1] = PR[90,1] + 77.686;
   1:  PR[91,2] = PR[90,2] + -6.758;
   1:L PR[91] R[100]mm/sec CNT100;
   1:  PR[91,1] = PR[90,1] + 77.359;
   1:  PR[91,2] = PR[90,2] + -7.213;
   1:L PR[91] R[100]mm/sec CNT100;
   1:  PR[91,1] = PR[90,1] + 76.818;
   1:  PR[91,2] = PR[90,2] + -7.885;
   1:L PR[91] R[100]mm/sec CNT100;
   1:  PR[91,1] = PR[90,1] + 76.285;
   1:  PR[91,2] = PR[90,2] + -8.530;
   1:L PR[91] R[100]mm/sec CNT100;
   1:  PR[91,1] = PR[90,1] + 75.844;
   1:  PR[91,2] = PR[90,2] + -9.001;
   1:L PR[91] R[100]mm/sec CNT100;
   1:  PR[91,1] = PR[90,1] + 74.729;
   1:  PR[91,2] = PR[90,2] + -10.082;
   1:L PR[91] R[100]mm/sec CNT100;
   1:  PR[91,1] = PR[90,1] + 74.081;
   1:  PR[91,2] = PR[90,2] + -10.612;
   1:L PR[91] R[100]mm/sec CNT100;
   1:  PR[91,1] = PR[90,1] + 72.971;
   1:  PR[91,2] = PR[90,2] + -11.466;
   1:L PR[91] R[100]mm/sec CNT100;
   1:  PR[91,1] = PR[90,1] + 72.303;
   1:  PR[91,2] = PR[90,2] + -11.838;
   1:L PR[91] R[100]mm/sec CNT100;
   1:  PR[91,1] = PR[90,1] + 71.882;
   1:  PR[91,2] = PR[90,2] + -12.038;
   1:L PR[91] R[100]mm/sec CNT100;
   1:  PR[91,1] = PR[90,1] + 71.525;
   1:  PR[91,2] = PR[90,2] + -12.278;
   1:L PR[91] R[100]mm/sec CNT100;
   1:  PR[91,1] = PR[90,1] + 70.737;
   1:  PR[91,2] = PR[90,2] + -12.685;
   1:L PR[91] R[100]mm/sec CNT100;
   1:  PR[91,1] = PR[90,1] + 70.086;
   1:  PR[91,2] = PR[90,2] + -12.921;
   1:L PR[91] R[100]mm/sec CNT100;
   1:  PR[91,1] = PR[90,1] + 69.618;
   1:  PR[91,2] = PR[90,2] + -13.050;
   1:L PR[91] R[100]mm/sec CNT100;
   1:  PR[91,1] = PR[90,1] + 68.601;
   1:  PR[91,2] = PR[90,2] + -13.473;
   1:L PR[91] R[100]mm/sec CNT100;
   1:  PR[91,1] = PR[90,1] + 67.392;
   1:  PR[91,2] = PR[90,2] + -13.783;
   1:L PR[91] R[100]mm/sec CNT100;
   1:  PR[91,1] = PR[90,1] + 65.754;
   1:  PR[91,2] = PR[90,2] + -13.971;
   1:L PR[91] R[100]mm/sec CNT100;
   1:  PR[91,1] = PR[90,1] + 64.629;
   1:  PR[91,2] = PR[90,2] + -14.016;
   1:L PR[91] R[100]mm/sec CNT100;
   1:  PR[91,1] = PR[90,1] + 64.093;
   1:  PR[91,2] = PR[90,2] + -14.021;
   1:L PR[91] R[100]mm/sec CNT100;
   1:  PR[91,1] = PR[90,1] + 63.001;
   1:  PR[91,2] = PR[90,2] + -13.995;
   1:L PR[91] R[100]mm/sec CNT100;
   1:  PR[91,1] = PR[90,1] + 62.537;
   1:  PR[91,2] = PR[90,2] + -13.946;
   1:L PR[91] R[100]mm/sec CNT100;
   1:  PR[91,1] = PR[90,1] + 61.971;
   1:  PR[91,2] = PR[90,2] + -13.922;
   1:L PR[91] R[100]mm/sec CNT100;
   1:  PR[91,1] = PR[90,1] + 60.516;
   1:  PR[91,2] = PR[90,2] + -13.743;
   1:L PR[91] R[100]mm/sec CNT100;
   1:  PR[91,1] = PR[90,1] + 59.434;
   1:  PR[91,2] = PR[90,2] + -13.429;
   1:L PR[91] R[100]mm/sec CNT100;
   1:  PR[91,1] = PR[90,1] + 58.906;
   1:  PR[91,2] = PR[90,2] + -13.113;
   1:L PR[91] R[100]mm/sec CNT100;
   1:  PR[91,1] = PR[90,1] + 58.668;
   1:  PR[91,2] = PR[90,2] + -13.083;
   1:L PR[91] R[100]mm/sec CNT100;
   1:  PR[91,1] = PR[90,1] + 58.157;
   1:  PR[91,2] = PR[90,2] + -12.854;
   1:L PR[91] R[100]mm/sec CNT100;
   1:  PR[91,1] = PR[90,1] + 57.217;
   1:  PR[91,2] = PR[90,2] + -12.634;
   1:L PR[91] R[100]mm/sec CNT100;
   1:  PR[91,1] = PR[90,1] + 56.487;
   1:  PR[91,2] = PR[90,2] + -12.145;
   1:L PR[91] R[100]mm/sec CNT100;
   1:  PR[91,1] = PR[90,1] + 56.469;
   1:  PR[91,2] = PR[90,2] + -12.142;
   1:L PR[91] R[100]mm/sec CNT100;
   1:  PR[91,1] = PR[90,1] + 55.927;
   1:  PR[91,2] = PR[90,2] + -11.756;
   1:L PR[91] R[100]mm/sec CNT100;
   1:  PR[91,1] = PR[90,1] + 54.995;
   1:  PR[91,2] = PR[90,2] + -11.420;
   1:L PR[91] R[100]mm/sec CNT100;
   1:  PR[91,1] = PR[90,1] + 54.532;
   1:  PR[91,2] = PR[90,2] + -10.860;
   1:L PR[91] R[100]mm/sec CNT100;
   1:  PR[91,1] = PR[90,1] + 54.517;
   1:  PR[91,2] = PR[90,2] + -10.838;
   1:L PR[91] R[100]mm/sec CNT100;
   1:  PR[91,1] = PR[90,1] + 54.474;
   1:  PR[91,2] = PR[90,2] + -10.825;
   1:L PR[91] R[100]mm/sec CNT100;
   1:  PR[91,1] = PR[90,1] + 53.806;
   1:  PR[91,2] = PR[90,2] + -10.449;
   1:L PR[91] R[100]mm/sec CNT100;
   1:  PR[91,1] = PR[90,1] + 53.260;
   1:  PR[91,2] = PR[90,2] + -9.840;
   1:L PR[91] R[100]mm/sec CNT100;
   1:  PR[91,1] = PR[90,1] + 52.660;
   1:  PR[91,2] = PR[90,2] + -9.355;
   1:L PR[91] R[100]mm/sec CNT100;
   1:  PR[91,1] = PR[90,1] + 52.170;
   1:  PR[91,2] = PR[90,2] + -8.759;
   1:L PR[91] R[100]mm/sec CNT100;
   1:  PR[91,1] = PR[90,1] + 51.563;
   1:  PR[91,2] = PR[90,2] + -8.201;
   1:L PR[91] R[100]mm/sec CNT100;
   1:  PR[91,1] = PR[90,1] + 51.167;
   1:  PR[91,2] = PR[90,2] + -7.531;
   1:L PR[91] R[100]mm/sec CNT100;
   1:  PR[91,1] = PR[90,1] + 51.165;
   1:  PR[91,2] = PR[90,2] + -7.523;
   1:L PR[91] R[100]mm/sec CNT100;
   1:  PR[91,1] = PR[90,1] + 50.548;
   1:  PR[91,2] = PR[90,2] + -6.999;
   1:L PR[91] R[100]mm/sec CNT100;
   1:  PR[91,1] = PR[90,1] + 50.257;
   1:  PR[91,2] = PR[90,2] + -6.112;
   1:L PR[91] R[100]mm/sec CNT100;
   1:  PR[91,1] = PR[90,1] + 49.950;
   1:  PR[91,2] = PR[90,2] + -5.746;
   1:L PR[91] R[100]mm/sec CNT100;
   1:  PR[91,1] = PR[90,1] + 49.920;
   1:  PR[91,2] = PR[90,2] + -5.726;
   1:L PR[91] R[100]mm/sec CNT100;
   1:  PR[91,1] = PR[90,1] + 49.889;
   1:  PR[91,2] = PR[90,2] + -5.673;
   1:L PR[91] R[100]mm/sec CNT100;
   1:  PR[91,1] = PR[90,1] + 49.808;
   1:  PR[91,2] = PR[90,2] + -5.578;
   1:L PR[91] R[100]mm/sec CNT100;
   1:  PR[91,1] = PR[90,1] + 49.797;
   1:  PR[91,2] = PR[90,2] + -5.519;
   1:L PR[91] R[100]mm/sec CNT100;
   1:  PR[91,1] = PR[90,1] + 49.359;
   1:  PR[91,2] = PR[90,2] + -4.779;
   1:L PR[91] R[100]mm/sec CNT100;
   1:  PR[91,1] = PR[90,1] + 49.212;
   1:  PR[91,2] = PR[90,2] + -4.237;
   1:L PR[91] R[100]mm/sec CNT100;
   1:  PR[91,1] = PR[90,1] + 49.142;
   1:  PR[91,2] = PR[90,2] + -3.863;
   1:L PR[91] R[100]mm/sec CNT100;
   1:  PR[91,1] = PR[90,1] + 48.868;
   1:  PR[91,2] = PR[90,2] + -3.352;
   1:L PR[91] R[100]mm/sec CNT100;
   1:  PR[91,1] = PR[90,1] + 48.850;
   1:  PR[91,2] = PR[90,2] + -3.207;
   1:L PR[91] R[100]mm/sec CNT100;
   1:  PR[91,1] = PR[90,1] + 48.751;
   1:  PR[91,2] = PR[90,2] + -3.073;
   1:L PR[91] R[100]mm/sec CNT100;
   1:  PR[91,1] = PR[90,1] + 48.447;
   1:  PR[91,2] = PR[90,2] + -2.466;
   1:L PR[91] R[100]mm/sec CNT100;
   1:  PR[91,1] = PR[90,1] + 48.406;
   1:  PR[91,2] = PR[90,2] + -2.172;
   1:L PR[91] R[100]mm/sec CNT100;
   1:  PR[91,1] = PR[90,1] + 48.224;
   1:  PR[91,2] = PR[90,2] + -1.467;
   1:L PR[91] R[100]mm/sec CNT100;
   1:  PR[91,1] = PR[90,1] + 48.121;
   1:  PR[91,2] = PR[90,2] + -0.489;
   1:L PR[91] R[100]mm/sec CNT100;
   1:  PR[91,1] = PR[90,1] + 48.040;
   1:  PR[91,2] = PR[90,2] + -0.012;
   1:L PR[91] R[100]mm/sec CNT100;
   1:  PR[91,1] = PR[90,1] + 48.020;
   1:  PR[91,2] = PR[90,2] + 0.509;
   1:L PR[91] R[100]mm/sec CNT100;
   1:  PR[91,1] = PR[90,1] + 47.950;
   1:  PR[91,2] = PR[90,2] + 1.044;
   1:L PR[91] R[100]mm/sec CNT100;
   1:  PR[91,1] = PR[90,1] + 47.941;
   1:  PR[91,2] = PR[90,2] + 1.508;
   1:L PR[91] R[100]mm/sec CNT100;
   1:  PR[91,1] = PR[90,1] + 47.902;
   1:  PR[91,2] = PR[90,2] + 2.111;
   1:L PR[91] R[100]mm/sec CNT100;
   1:  PR[91,1] = PR[90,1] + 47.880;
   1:  PR[91,2] = PR[90,2] + 4.183;
   1:L PR[91] R[100]mm/sec CNT100;
   1:  PR[91,1] = PR[90,1] + 47.877;
   1:  PR[91,2] = PR[90,2] + 23.385;
   1:L PR[91] R[100]mm/sec CNT100;
   1:  PR[91,1] = PR[90,1] + 47.836;
   1:  PR[91,2] = PR[90,2] + 24.514;
   1:L PR[91] R[100]mm/sec CNT100;
   1:  PR[91,1] = PR[90,1] + 47.730;
   1:  PR[91,2] = PR[90,2] + 24.937;
   1:L PR[91] R[100]mm/sec CNT100;
   1:  PR[91,1] = PR[90,1] + 47.704;
   1:  PR[91,2] = PR[90,2] + 24.971;
   1:L PR[91] R[100]mm/sec CNT100;
   1:  PR[91,1] = PR[90,1] + 47.365;
   1:  PR[91,2] = PR[90,2] + 25.831;
   1:L PR[91] R[100]mm/sec CNT100;
   1:  PR[91,1] = PR[90,1] + 47.319;
   1:  PR[91,2] = PR[90,2] + 26.107;
   1:L PR[91] R[100]mm/sec CNT100;
   1:  PR[91,1] = PR[90,1] + 47.215;
   1:  PR[91,2] = PR[90,2] + 26.455;
   1:L PR[91] R[100]mm/sec CNT100;
   1:  PR[91,1] = PR[90,1] + 47.044;
   1:  PR[91,2] = PR[90,2] + 26.768;
   1:L PR[91] R[100]mm/sec CNT100;
   1:  PR[91,1] = PR[90,1] + 46.544;
   1:  PR[91,2] = PR[90,2] + 27.293;
   1:L PR[91] R[100]mm/sec CNT100;
   1:  PR[91,1] = PR[90,1] + 46.279;
   1:  PR[91,2] = PR[90,2] + 27.751;
   1:L PR[91] R[100]mm/sec CNT100;
   1:  PR[91,1] = PR[90,1] + 45.809;
   1:  PR[91,2] = PR[90,2] + 28.025;
   1:L PR[91] R[100]mm/sec CNT100;
   1:  PR[92] = PR[91];
   1:  PR[92,3] = PR[92,3] + R[101];
   1:J PR[92] R[102]% CNT100;
   1:  PR[91,1] = PR[90,1] + 43.628;
   1:  PR[91,2] = PR[90,2] + 26.421;
   1:  PR[92] = PR[91];
   1:  PR[92,3] = PR[92,3] + R[101];
   1:J PR[92] R[102]% CNT100;
   1:L PR[91] 100mm/sec CNT100 RampTo R[100];
   1:  PR[91,1] = PR[90,1] + 39.805;
   1:  PR[91,2] = PR[90,2] + 22.599;
   1:L PR[91] R[100]mm/sec CNT100;
   1:  PR[91,2] = PR[90,2] + 22.396;
   1:L PR[91] R[100]mm/sec CNT100;
   1:  PR[91,2] = PR[90,2] + 18.356;
   1:L PR[91] R[100]mm/sec CNT100;
   1:  PR[91,1] = PR[90,1] + 45.308;
   1:  PR[91,2] = PR[90,2] + 23.859;
   1:L PR[91] R[100]mm/sec CNT100;
   1:  PR[91,1] = PR[90,1] + 45.327;
   1:  PR[91,2] = PR[90,2] + 23.338;
   1:L PR[91] R[100]mm/sec CNT100;
   1:  PR[91,1] = PR[90,1] + 45.328;
   1:  PR[91,2] = PR[90,2] + 19.636;
   1:L PR[91] R[100]mm/sec CNT100;
   1:  PR[91,1] = PR[90,1] + 39.805;
   1:  PR[91,2] = PR[90,2] + 14.113;
   1:L PR[91] R[100]mm/sec CNT100;
   1:  PR[91,2] = PR[90,2] + 9.871;
   1:L PR[91] R[100]mm/sec CNT100;
   1:  PR[91,1] = PR[90,1] + 45.328;
   1:  PR[91,2] = PR[90,2] + 15.394;
   1:L PR[91] R[100]mm/sec CNT100;
   1:  PR[91,1] = PR[90,1] + 45.329;
   1:  PR[91,2] = PR[90,2] + 11.152;
   1:L PR[91] R[100]mm/sec CNT100;
   1:  PR[91,1] = PR[90,1] + 39.806;
   1:  PR[91,2] = PR[90,2] + 5.629;
   1:L PR[91] R[100]mm/sec CNT100;
   1:  PR[91,2] = PR[90,2] + 3.190;
   1:L PR[91] R[100]mm/sec CNT100;
   1:  PR[91,1] = PR[90,1] + 39.813;
   1:  PR[91,2] = PR[90,2] + 2.035;
   1:L PR[91] R[100]mm/sec CNT100;
   1:  PR[91,1] = PR[90,1] + 39.830;
   1:  PR[91,2] = PR[90,2] + 1.410;
   1:L PR[91] R[100]mm/sec CNT100;
   1:  PR[91,1] = PR[90,1] + 45.330;
   1:  PR[91,2] = PR[90,2] + 6.910;
   1:L PR[91] R[100]mm/sec CNT100;
   1:  PR[91,2] = PR[90,2] + 4.169;
   1:L PR[91] R[100]mm/sec CNT100;
   1:  PR[91,1] = PR[90,1] + 45.346;
   1:  PR[91,2] = PR[90,2] + 2.684;
   1:L PR[91] R[100]mm/sec CNT100;
   1:  PR[91,1] = PR[90,1] + 40.316;
   1:  PR[91,2] = PR[90,2] + -2.347;
   1:L PR[91] R[100]mm/sec CNT100;
   1:  PR[91,1] = PR[90,1] + 40.326;
   1:  PR[91,2] = PR[90,2] + -2.506;
   1:L PR[91] R[100]mm/sec CNT100;
   1:  PR[91,1] = PR[90,1] + 40.374;
   1:  PR[91,2] = PR[90,2] + -2.884;
   1:L PR[91] R[100]mm/sec CNT100;
   1:  PR[91,1] = PR[90,1] + 40.453;
   1:  PR[91,2] = PR[90,2] + -3.331;
   1:L PR[91] R[100]mm/sec CNT100;
   1:  PR[91,1] = PR[90,1] + 40.478;
   1:  PR[91,2] = PR[90,2] + -3.564;
   1:L PR[91] R[100]mm/sec CNT100;
   1:  PR[91,1] = PR[90,1] + 40.611;
   1:  PR[91,2] = PR[90,2] + -4.000;
   1:L PR[91] R[100]mm/sec CNT100;
   1:  PR[91,1] = PR[90,1] + 40.980;
   1:  PR[91,2] = PR[90,2] + -4.715;
   1:L PR[91] R[100]mm/sec CNT100;
   1:  PR[91,1] = PR[90,1] + 41.007;
   1:  PR[91,2] = PR[90,2] + -5.007;
   1:L PR[91] R[100]mm/sec CNT100;
   1:  PR[91,1] = PR[90,1] + 41.232;
   1:  PR[91,2] = PR[90,2] + -5.602;
   1:L PR[91] R[100]mm/sec CNT100;
   1:  PR[91,1] = PR[90,1] + 41.241;
   1:  PR[91,2] = PR[90,2] + -5.664;
   1:L PR[91] R[100]mm/sec CNT100;
   1:  PR[91,1] = PR[90,1] + 45.639;
   1:  PR[91,2] = PR[90,2] + -1.266;
   1:L PR[91] R[100]mm/sec CNT100;
   1:  PR[91,1] = PR[90,1] + 45.707;
   1:  PR[91,2] = PR[90,2] + -1.922;
   1:L PR[91] R[100]mm/sec CNT100;
   1:  PR[91,1] = PR[90,1] + 45.901;
   1:  PR[91,2] = PR[90,2] + -2.668;
   1:L PR[91] R[100]mm/sec CNT100;
   1:  PR[91,1] = PR[90,1] + 45.979;
   1:  PR[91,2] = PR[90,2] + -3.233;
   1:L PR[91] R[100]mm/sec CNT100;
   1:  PR[91,1] = PR[90,1] + 46.383;
   1:  PR[91,2] = PR[90,2] + -4.039;
   1:L PR[91] R[100]mm/sec CNT100;
   1:  PR[91,1] = PR[90,1] + 46.395;
   1:  PR[91,2] = PR[90,2] + -4.135;
   1:L PR[91] R[100]mm/sec CNT100;
   1:  PR[91,1] = PR[90,1] + 46.610;
   1:  PR[91,2] = PR[90,2] + -4.537;
   1:L PR[91] R[100]mm/sec CNT100;
   1:  PR[91,1] = PR[90,1] + 42.571;
   1:  PR[91,2] = PR[90,2] + -8.576;
   1:L PR[91] R[100]mm/sec CNT100;
   1:  PR[91,1] = PR[90,1] + 42.832;
   1:  PR[91,2] = PR[90,2] + -8.807;
   1:L PR[91] R[100]mm/sec CNT100;
   1:  PR[91,1] = PR[90,1] + 42.985;
   1:  PR[91,2] = PR[90,2] + -9.718;
   1:L PR[91] R[100]mm/sec CNT100;
   1:  PR[91,1] = PR[90,1] + 43.056;
   1:  PR[91,2] = PR[90,2] + -9.862;
   1:L PR[91] R[100]mm/sec CNT100;
   1:  PR[91,1] = PR[90,1] + 43.082;
   1:  PR[91,2] = PR[90,2] + -9.919;
   1:L PR[91] R[100]mm/sec CNT100;
   1:  PR[91,1] = PR[90,1] + 43.826;
   1:  PR[91,2] = PR[90,2] + -10.546;
   1:L PR[91] R[100]mm/sec CNT100;
   1:  PR[91,1] = PR[90,1] + 44.024;
   1:  PR[91,2] = PR[90,2] + -11.366;
   1:L PR[91] R[100]mm/sec CNT100;
   1:  PR[91,1] = PR[90,1] + 47.963;
   1:  PR[91,2] = PR[90,2] + -7.427;
   1:L PR[91] R[100]mm/sec CNT100;
   1:  PR[91,1] = PR[90,1] + 48.017;
   1:  PR[91,2] = PR[90,2] + -7.518;
   1:L PR[91] R[100]mm/sec CNT100;
   1:  PR[91,1] = PR[90,1] + 48.039;
   1:  PR[91,2] = PR[90,2] + -7.533;
   1:L PR[91] R[100]mm/sec CNT100;
   1:  PR[91,1] = PR[90,1] + 48.349;
   1:  PR[91,2] = PR[90,2] + -8.476;
   1:L PR[91] R[100]mm/sec CNT100;
   1:  PR[91,1] = PR[90,1] + 49.182;
   1:  PR[91,2] = PR[90,2] + -9.184;
   1:L PR[91] R[100]mm/sec CNT100;
   1:  PR[91,1] = PR[90,1] + 49.559;
   1:  PR[91,2] = PR[90,2] + -9.823;
   1:L PR[91] R[100]mm/sec CNT100;
   1:  PR[91,1] = PR[90,1] + 49.690;
   1:  PR[91,2] = PR[90,2] + -9.943;
   1:L PR[91] R[100]mm/sec CNT100;
   1:  PR[91,1] = PR[90,1] + 45.954;
   1:  PR[91,2] = PR[90,2] + -13.679;
   1:L PR[91] R[100]mm/sec CNT100;
   1:  PR[91,1] = PR[90,1] + 46.427;
   1:  PR[91,2] = PR[90,2] + -13.933;
   1:L PR[91] R[100]mm/sec CNT100;
   1:  PR[91,1] = PR[90,1] + 46.667;
   1:  PR[91,2] = PR[90,2] + -14.512;
   1:L PR[91] R[100]mm/sec CNT100;
   1:  PR[91,1] = PR[90,1] + 47.272;
   1:  PR[91,2] = PR[90,2] + -14.784;
   1:L PR[91] R[100]mm/sec CNT100;
   1:  PR[91,1] = PR[90,1] + 47.558;
   1:  PR[91,2] = PR[90,2] + -15.413;
   1:L PR[91] R[100]mm/sec CNT100;
   1:  PR[91,1] = PR[90,1] + 48.059;
   1:  PR[91,2] = PR[90,2] + -15.626;
   1:L PR[91] R[100]mm/sec CNT100;
   1:  PR[91,1] = PR[90,1] + 48.130;
   1:  PR[91,2] = PR[90,2] + -15.746;
   1:L PR[91] R[100]mm/sec CNT100;
   1:  PR[91,1] = PR[90,1] + 51.821;
   1:  PR[91,2] = PR[90,2] + -12.054;
   1:L PR[91] R[100]mm/sec CNT100;
   1:  PR[91,1] = PR[90,1] + 52.188;
   1:  PR[91,2] = PR[90,2] + -12.464;
   1:L PR[91] R[100]mm/sec CNT100;
   1:  PR[91,1] = PR[90,1] + 52.865;
   1:  PR[91,2] = PR[90,2] + -12.846;
   1:L PR[91] R[100]mm/sec CNT100;
   1:  PR[91,1] = PR[90,1] + 53.475;
   1:  PR[91,2] = PR[90,2] + -13.582;
   1:L PR[91] R[100]mm/sec CNT100;
   1:  PR[91,1] = PR[90,1] + 54.255;
   1:  PR[91,2] = PR[90,2] + -13.863;
   1:L PR[91] R[100]mm/sec CNT100;
   1:  PR[91,1] = PR[90,1] + 50.326;
   1:  PR[91,2] = PR[90,2] + -17.792;
   1:L PR[91] R[100]mm/sec CNT100;
   1:  PR[91,1] = PR[90,1] + 50.528;
   1:  PR[91,2] = PR[90,2] + -17.969;
   1:L PR[91] R[100]mm/sec CNT100;
   1:  PR[91,1] = PR[90,1] + 50.630;
   1:  PR[91,2] = PR[90,2] + -18.044;
   1:L PR[91] R[100]mm/sec CNT100;
   1:  PR[91,1] = PR[90,1] + 51.406;
   1:  PR[91,2] = PR[90,2] + -18.254;
   1:L PR[91] R[100]mm/sec CNT100;
   1:  PR[91,1] = PR[90,1] + 52.133;
   1:  PR[91,2] = PR[90,2] + -19.009;
   1:L PR[91] R[100]mm/sec CNT100;
   1:  PR[91,1] = PR[90,1] + 52.197;
   1:  PR[91,2] = PR[90,2] + -19.041;
   1:L PR[91] R[100]mm/sec CNT100;
   1:  PR[91,1] = PR[90,1] + 52.230;
   1:  PR[91,2] = PR[90,2] + -19.056;
   1:L PR[91] R[100]mm/sec CNT100;
   1:  PR[91,1] = PR[90,1] + 53.072;
   1:  PR[91,2] = PR[90,2] + -19.209;
   1:L PR[91] R[100]mm/sec CNT100;
   1:  PR[91,1] = PR[90,1] + 53.113;
   1:  PR[91,2] = PR[90,2] + -19.248;
   1:L PR[91] R[100]mm/sec CNT100;
   1:  PR[91,1] = PR[90,1] + 57.129;
   1:  PR[91,2] = PR[90,2] + -15.232;
   1:L PR[91] R[100]mm/sec CNT100;
   1:  PR[91,1] = PR[90,1] + 57.337;
   1:  PR[91,2] = PR[90,2] + -15.281;
   1:L PR[91] R[100]mm/sec CNT100;
   1:  PR[91,1] = PR[90,1] + 57.970;
   1:  PR[91,2] = PR[90,2] + -15.565;
   1:L PR[91] R[100]mm/sec CNT100;
   1:  PR[91,1] = PR[90,1] + 58.054;
   1:  PR[91,2] = PR[90,2] + -15.575;
   1:L PR[91] R[100]mm/sec CNT100;
   1:  PR[91,1] = PR[90,1] + 58.407;
   1:  PR[91,2] = PR[90,2] + -15.787;
   1:L PR[91] R[100]mm/sec CNT100;
   1:  PR[91,1] = PR[90,1] + 60.002;
   1:  PR[91,2] = PR[90,2] + -16.249;
   1:L PR[91] R[100]mm/sec CNT100;
   1:  PR[91,1] = PR[90,1] + 60.316;
   1:  PR[91,2] = PR[90,2] + -16.288;
   1:L PR[91] R[100]mm/sec CNT100;
   1:  PR[91,1] = PR[90,1] + 55.845;
   1:  PR[91,2] = PR[90,2] + -20.758;
   1:L PR[91] R[100]mm/sec CNT100;
   1:  PR[91,1] = PR[90,1] + 56.380;
   1:  PR[91,2] = PR[90,2] + -20.856;
   1:L PR[91] R[100]mm/sec CNT100;
   1:  PR[91,1] = PR[90,1] + 56.877;
   1:  PR[91,2] = PR[90,2] + -21.011;
   1:L PR[91] R[100]mm/sec CNT100;
   1:  PR[91,1] = PR[90,1] + 57.247;
   1:  PR[91,2] = PR[90,2] + -21.048;
   1:L PR[91] R[100]mm/sec CNT100;
   1:  PR[91,1] = PR[90,1] + 58.250;
   1:  PR[91,2] = PR[90,2] + -21.493;
   1:L PR[91] R[100]mm/sec CNT100;
   1:  PR[91,1] = PR[90,1] + 58.528;
   1:  PR[91,2] = PR[90,2] + -21.589;
   1:L PR[91] R[100]mm/sec CNT100;
   1:  PR[91,1] = PR[90,1] + 58.704;
   1:  PR[91,2] = PR[90,2] + -21.607;
   1:L PR[91] R[100]mm/sec CNT100;
   1:  PR[91,1] = PR[90,1] + 59.141;
   1:  PR[91,2] = PR[90,2] + -21.700;
   1:L PR[91] R[100]mm/sec CNT100;
   1:  PR[91,1] = PR[90,1] + 59.145;
   1:  PR[91,2] = PR[90,2] + -21.701;
   1:L PR[91] R[100]mm/sec CNT100;
   1:  PR[91,1] = PR[90,1] + 64.276;
   1:  PR[91,2] = PR[90,2] + -16.570;
   1:L PR[91] R[100]mm/sec CNT100;
   1:  PR[91,1] = PR[90,1] + 64.691;
   1:  PR[91,2] = PR[90,2] + -16.566;
   1:L PR[91] R[100]mm/sec CNT100;
   1:  PR[91,1] = PR[90,1] + 65.952;
   1:  PR[91,2] = PR[90,2] + -16.515;
   1:L PR[91] R[100]mm/sec CNT100;
   1:  PR[91,1] = PR[90,1] + 67.856;
   1:  PR[91,2] = PR[90,2] + -16.296;
   1:L PR[91] R[100]mm/sec CNT100;
   1:  PR[91,1] = PR[90,1] + 69.115;
   1:  PR[91,2] = PR[90,2] + -15.974;
   1:L PR[91] R[100]mm/sec CNT100;
   1:  PR[91,1] = PR[90,1] + 62.971;
   1:  PR[91,2] = PR[90,2] + -22.118;
   1:L PR[91] R[100]mm/sec CNT100;
   1:  PR[91,1] = PR[90,1] + 63.287;
   1:  PR[91,2] = PR[90,2] + -22.143;
   1:L PR[91] R[100]mm/sec CNT100;
   1:  PR[91,1] = PR[90,1] + 64.103;
   1:  PR[91,2] = PR[90,2] + -22.166;
   1:L PR[91] R[100]mm/sec CNT100;
   1:  PR[91,1] = PR[90,1] + 64.893;
   1:  PR[91,2] = PR[90,2] + -22.143;
   1:L PR[91] R[100]mm/sec CNT100;
   1:  PR[91,1] = PR[90,1] + 65.812;
   1:  PR[91,2] = PR[90,2] + -22.072;
   1:L PR[91] R[100]mm/sec CNT100;
   1:  PR[91,1] = PR[90,1] + 66.837;
   1:  PR[91,2] = PR[90,2] + -21.971;
   1:L PR[91] R[100]mm/sec CNT100;
   1:  PR[91,1] = PR[90,1] + 67.433;
   1:  PR[91,2] = PR[90,2] + -21.898;
   1:L PR[91] R[100]mm/sec CNT100;
   1:  PR[91,1] = PR[90,1] + 88.080;
   1:  PR[91,2] = PR[90,2] + -1.252;
   1:L PR[91] R[100]mm/sec CNT100;
   1:  PR[91,1] = PR[90,1] + 88.056;
   1:  PR[91,2] = PR[90,2] + -1.410;
   1:L PR[91] R[100]mm/sec CNT100;
   1:  PR[91,1] = PR[90,1] + 88.045;
   1:  PR[91,2] = PR[90,2] + -1.543;
   1:L PR[91] R[100]mm/sec CNT100;
   1:  PR[91,1] = PR[90,1] + 87.922;
   1:  PR[91,2] = PR[90,2] + -2.249;
   1:L PR[91] R[100]mm/sec CNT100;
   1:  PR[91,1] = PR[90,1] + 87.793;
   1:  PR[91,2] = PR[90,2] + -3.128;
   1:L PR[91] R[100]mm/sec CNT100;
   1:  PR[91,1] = PR[90,1] + 87.616;
   1:  PR[91,2] = PR[90,2] + -3.853;
   1:L PR[91] R[100]mm/sec CNT100;
   1:  PR[91,1] = PR[90,1] + 87.601;
   1:  PR[91,2] = PR[90,2] + -4.012;
   1:L PR[91] R[100]mm/sec CNT100;
   1:  PR[91,1] = PR[90,1] + 87.387;
   1:  PR[91,2] = PR[90,2] + -4.599;
   1:L PR[91] R[100]mm/sec CNT100;
   1:  PR[91,1] = PR[90,1] + 87.029;
   1:  PR[91,2] = PR[90,2] + -5.684;
   1:L PR[91] R[100]mm/sec CNT100;
   1:  PR[91,1] = PR[90,1] + 86.797;
   1:  PR[91,2] = PR[90,2] + -6.406;
   1:L PR[91] R[100]mm/sec CNT100;
   1:  PR[91,1] = PR[90,1] + 86.759;
   1:  PR[91,2] = PR[90,2] + -6.578;
   1:L PR[91] R[100]mm/sec CNT100;
   1:  PR[91,1] = PR[90,1] + 86.520;
   1:  PR[91,2] = PR[90,2] + -7.054;
   1:L PR[91] R[100]mm/sec CNT100;
   1:  PR[91,1] = PR[90,1] + 73.228;
   1:  PR[91,2] = PR[90,2] + -20.346;
   1:L PR[91] R[100]mm/sec CNT100;
   1:  PR[92] = PR[91];
   1:  PR[92,3] = PR[92,3] + R[101];
   1:J PR[92] R[102]% CNT100;
   1:  PR[91,1] = PR[90,1] + 82.299;
   1:  PR[91,2] = PR[90,2] + -2.790;
   1:  PR[92] = PR[91];
   1:  PR[92,3] = PR[92,3] + R[101];
   1:J PR[92] R[102]% CNT100;
   1:L PR[91] 100mm/sec CNT100 RampTo R[100];
   1:  PR[91,1] = PR[90,1] + 88.450;
   1:  PR[91,2] = PR[90,2] + 3.362;
   1:L PR[91] R[100]mm/sec CNT100;
   1:  PR[91,1] = PR[90,1] + 88.452;
   1:  PR[91,2] = PR[90,2] + 7.606;
   1:L PR[91] R[100]mm/sec CNT100;
   1:  PR[91,1] = PR[90,1] + 82.874;
   1:  PR[91,2] = PR[90,2] + 2.027;
   1:L PR[91] R[100]mm/sec CNT100;
   1:  PR[91,1] = PR[90,1] + 82.890;
   1:  PR[91,2] = PR[90,2] + 3.148;
   1:L PR[91] R[100]mm/sec CNT100;
   1:  PR[91,1] = PR[90,1] + 82.891;
   1:  PR[91,2] = PR[90,2] + 6.287;
   1:L PR[91] R[100]mm/sec CNT100;
   1:  PR[91,1] = PR[90,1] + 88.454;
   1:  PR[91,2] = PR[90,2] + 11.850;
   1:L PR[91] R[100]mm/sec CNT100;
   1:  PR[91,1] = PR[90,1] + 88.455;
   1:  PR[91,2] = PR[90,2] + 16.094;
   1:L PR[91] R[100]mm/sec CNT100;
   1:  PR[91,1] = PR[90,1] + 82.891;
   1:  PR[91,2] = PR[90,2] + 10.530;
   1:L PR[91] R[100]mm/sec CNT100;
   1:  PR[91,1] = PR[90,1] + 82.892;
   1:  PR[91,2] = PR[90,2] + 14.773;
   1:L PR[91] R[100]mm/sec CNT100;
   1:  PR[91,1] = PR[90,1] + 88.457;
   1:  PR[91,2] = PR[90,2] + 20.339;
   1:L PR[91] R[100]mm/sec CNT100;
   1:  PR[91,1] = PR[90,1] + 88.458;
   1:  PR[91,2] = PR[90,2] + 22.386;
   1:L PR[91] R[100]mm/sec CNT100;
   1:  PR[91,1] = PR[90,1] + 88.448;
   1:  PR[91,2] = PR[90,2] + 23.526;
   1:L PR[91] R[100]mm/sec CNT100;
   1:  PR[91,1] = PR[90,1] + 88.425;
   1:  PR[91,2] = PR[90,2] + 23.905;
   1:L PR[91] R[100]mm/sec CNT100;
   1:  PR[91,1] = PR[90,1] + 88.313;
   1:  PR[91,2] = PR[90,2] + 24.280;
   1:L PR[91] R[100]mm/sec CNT100;
   1:  PR[91,1] = PR[90,1] + 88.294;
   1:  PR[91,2] = PR[90,2] + 24.374;
   1:L PR[91] R[100]mm/sec CNT100;
   1:  PR[91,1] = PR[90,1] + 88.283;
   1:  PR[91,2] = PR[90,2] + 24.407;
   1:L PR[91] R[100]mm/sec CNT100;
   1:  PR[91,1] = PR[90,1] + 82.892;
   1:  PR[91,2] = PR[90,2] + 19.016;
   1:L PR[91] R[100]mm/sec CNT100;
   1:  PR[91,2] = PR[90,2] + 22.393;
   1:L PR[91] R[100]mm/sec CNT100;
   1:  PR[91,1] = PR[90,1] + 82.896;
   1:  PR[91,2] = PR[90,2] + 23.263;
   1:L PR[91] R[100]mm/sec CNT100;
   1:  PR[91,1] = PR[90,1] + 86.263;
   1:  PR[91,2] = PR[90,2] + 26.630;
   1:L PR[91] R[100]mm/sec CNT100  Weld End[1,5.0,0.2s];
   1:  PR[92] = PR[91];
   1:  PR[92,3] = PR[92,3] + 100;
   1:J PR[92] R[102]% CNT100;
   1:  WAIT   5.00(sec);
   1:  CALL HOME_ALL;
/POS
/END
